LIN {X 0,Y 156.814,Z 593.588,A -85,B 0,C 180,E1 -25031.921,E2 -25031.921} C_VEL
LIN {X 0,Y 150.311,Z 600.724,A -85,B 0,C 180,E1 -25035.498,E2 -25035.498} C_VEL
LIN {X 0,Y 145.203,Z 605.623,A -85,B 0,C 180,E1 -25038.8,E2 -25038.8} C_VEL
LIN {X 0,Y 138.955,Z 610.891,A -85,B 0,C 180,E1 -25043.868,E2 -25043.868} C_VEL
LIN {X 0,Y 135.035,Z 613.658,A -85,B 0,C 180,E1 -25047.932,E2 -25047.932} C_VEL
LIN {X 0,Y 131.858,Z 615.519,A -85,B 0,C 180,E1 -25052.209,E2 -25052.209} C_VEL
LIN {X 0,Y 129.32,Z 616.538,A -85,B 0,C 180,E1 -25056.713,E2 -25056.713} C_VEL
LIN {X 0,Y 127.481,Z 616.693,A -85,B 0,C 180,E1 -25061.42,E2 -25061.42} C_VEL
LIN {X 0,Y 126.047,Z 615.481,A -85,B 0,C 180,E1 -25067.999,E2 -25067.999} C_VEL
LIN {X 0,Y 125.854,Z 612.811,A -85,B 0,C 180,E1 -25074.097,E2 -25074.097} C_VEL
LIN {X 0,Y 126.43,Z 610.019,A -85,B 0,C 180,E1 -25078.395,E2 -25078.395} C_VEL
LIN {X 0,Y 127.613,Z 605.119,A -85,B 0,C 180,E1 -25083.855,E2 -25083.855} C_VEL
LIN {X 0,Y 129.275,Z 599.296,A -85,B 0,C 180,E1 -25088.733,E2 -25088.733} C_VEL
LIN {X 0,Y 131.792,Z 591.532,A -85,B 0,C 180,E1 -25093.717,E2 -25093.717} C_VEL
LIN {X 0,Y 134.655,Z 582.904,A -85,B 0,C 180,E1 -25097.946,E2 -25097.946} C_VEL
LIN {X 0,Y 137.776,Z 573.446,A -85,B 0,C 180,E1 -25101.563,E2 -25101.563} C_VEL
LIN {X 0,Y 140.914,Z 563.091,A -85,B 0,C 180,E1 -25104.647,E2 -25104.647} C_VEL
LIN {X 0,Y 143.932,Z 551.949,A -85,B 0,C 180,E1 -25107.198,E2 -25107.198} C_VEL
LIN {X 0,Y 146.787,Z 539.398,A -85,B 0,C 180,E1 -25109.38,E2 -25109.38} C_VEL
LIN {X 0,Y 149.013,Z 526.448,A -85,B 0,C 180,E1 -25111.001,E2 -25111.001} C_VEL
LIN {X 0,Y 150.791,Z 512.614,A -85,B 0,C 180,E1 -25112.147,E2 -25112.147} C_VEL
LIN {X 0,Y 154.321,Z 464.5,A -85,B 0,C 180,E1 -25114.472,E2 -25114.472} C_VEL
LIN {X 0,Y 151.514,Z 456.717,A -85,B 0,C 180,E1 -25115.652,E2 -25115.652} C_VEL
LIN {X 0,Y 145.99,Z 443.962,A -85,B 0,C 180,E1 -25117.978,E2 -25117.978} C_VEL
LIN {X 0,Y 136.343,Z 427.063,A -85,B 0,C 180,E1 -25122.154,E2 -25122.154} C_VEL
LIN {X 0,Y 133.91,Z 423.355,A -85,B 0,C 180,E1 -25123.296,E2 -25123.296} C_VEL
LIN {X 0,Y 131.689,Z 419.888,A -85,B 0,C 180,E1 -25124.377,E2 -25124.377} C_VEL
LIN {X 0,Y 129.747,Z 417.326,A -85,B 0,C 180,E1 -25125.327,E2 -25125.327} C_VEL
LIN {X 0,Y 129.207,Z 415.394,A -85,B 0,C 180,E1 -25125.777,E2 -25125.777} C_VEL
LIN {X 0,Y 129.159,Z 415.379,A -85,B 0,C 180,E1 -25129.051,E2 -25129.051} C_VEL
LIN {X 0,Y 129.107,Z 415.403,A -85,B 0,C 180,E1 -25132.394,E2 -25132.394} C_VEL
LIN {X 0,Y 129.12,Z 415.555,A -85,B 0,C 180,E1 -25138.437,E2 -25138.437} C_VEL
LIN {X 0,Y 141.163,Z 449.103,A -85,B 0,C 180,E1 -25142.935,E2 -25142.935} C_VEL
LIN {X 0,Y 142.539,Z 453.928,A -85,B 0,C 180,E1 -25143.477,E2 -25143.477} C_VEL
LIN {X 0,Y 138.064,Z 512.835,A -85,B 0,C 180,E1 -25147.853,E2 -25147.853} C_VEL
LIN {X 0,Y 136.81,Z 526.19,A -85,B 0,C 180,E1 -25149.363,E2 -25149.363} C_VEL
LIN {X 0,Y 135.038,Z 539.905,A -85,B 0,C 180,E1 -25151.57,E2 -25151.57} C_VEL
LIN {X 0,Y 133.267,Z 551.828,A -85,B 0,C 180,E1 -25154.123,E2 -25154.123} C_VEL
LIN {X 0,Y 131.313,Z 563.456,A -85,B 0,C 180,E1 -25157.328,E2 -25157.328} C_VEL
LIN {X 0,Y 129.648,Z 573.756,A -85,B 0,C 180,E1 -25160.937,E2 -25160.937} C_VEL
LIN {X 0,Y 128.192,Z 583.694,A -85,B 0,C 180,E1 -25165.314,E2 -25165.314} C_VEL
LIN {X 0,Y 127.16,Z 592.452,A -85,B 0,C 180,E1 -25170.17,E2 -25170.17} C_VEL
LIN {X 0,Y 126.587,Z 598.713,A -85,B 0,C 180,E1 -25174.515,E2 -25174.515} C_VEL
LIN {X 0,Y 126.242,Z 603.697,A -85,B 0,C 180,E1 -25178.785,E2 -25178.785} C_VEL
LIN {X 0,Y 126.536,Z 608.396,A -85,B 0,C 180,E1 -25183.876,E2 -25183.876} C_VEL
LIN {X 0,Y 127.673,Z 611.966,A -85,B 0,C 180,E1 -25188.891,E2 -25188.891} C_VEL
LIN {X 0,Y 129.652,Z 614.508,A -85,B 0,C 180,E1 -25193.776,E2 -25193.776} C_VEL
LIN {X 0,Y 133.699,Z 616.42,A -85,B 0,C 180,E1 -25200,E2 -25200} C_VEL
LIN {X 0,Y 136.366,Z 616.802,A -85,B 0,C 180,E1 -25202.954,E2 -25202.954} C_VEL
LIN {X 0,Y 141.861,Z 616.494,A -85,B 0,C 180,E1 -25207.798,E2 -25207.798} C_VEL
LIN {X 0,Y 146.515,Z 615.477,A -85,B 0,C 180,E1 -25211.062,E2 -25211.062} C_VEL
LIN {X 0,Y 152.429,Z 613.559,A -85,B 0,C 180,E1 -25214.495,E2 -25214.495} C_VEL
LIN {X 0,Y 159.649,Z 610.415,A -85,B 0,C 180,E1 -25217.948,E2 -25217.948} C_VEL
LIN {X 0,Y 167.163,Z 606.309,A -85,B 0,C 180,E1 -25220.938,E2 -25220.938} C_VEL
LIN {X 0,Y 175.327,Z 600.967,A -85,B 0,C 180,E1 -25223.631,E2 -25223.631} C_VEL
LIN {X 0,Y 183.895,Z 594.271,A -85,B 0,C 180,E1 -25226.072,E2 -25226.072} C_VEL
LIN {X 0,Y 191.851,Z 586.996,A -85,B 0,C 180,E1 -25228.006,E2 -25228.006} C_VEL
LIN {X 0,Y 200.929,Z 577.067,A -85,B 0,C 180,E1 -25229.954,E2 -25229.954} C_VEL
LIN {X 0,Y 208.869,Z 566.785,A -85,B 0,C 180,E1 -25231.436,E2 -25231.436} C_VEL
LIN {X 0,Y 215.861,Z 555.807,A -85,B 0,C 180,E1 -25232.604,E2 -25232.604} C_VEL
LIN {X 0,Y 222.008,Z 544.013,A -85,B 0,C 180,E1 -25233.573,E2 -25233.573} C_VEL
LIN {X 0,Y 222.564,Z 542.783,A -85,B 0,C 180,E1 -25233.661,E2 -25233.661} C_VEL
LIN {X 0,Y 222.26,Z 543.527,A -85,B 0,C 180,E1 -25234.024,E2 -25234.024} C_VEL
LIN {X 0,Y 216.111,Z 555.561,A -85,B 0,C 180,E1 -25234.806,E2 -25234.806} C_VEL
LIN {X 0,Y 209.059,Z 566.785,A -85,B 0,C 180,E1 -25235.81,E2 -25235.81} C_VEL
LIN {X 0,Y 202.204,Z 576.047,A -85,B 0,C 180,E1 -25236.931,E2 -25236.931} C_VEL
LIN {X 0,Y 193.406,Z 586.164,A -85,B 0,C 180,E1 -25238.628,E2 -25238.628} C_VEL
LIN {X 0,Y 184.852,Z 594.451,A -85,B 0,C 180,E1 -25240.506,E2 -25240.506} C_VEL
LIN {X 0,Y 176.702,Z 601.316,A -85,B 0,C 180,E1 -25242.63,E2 -25242.63} C_VEL
LIN {X 0,Y 168.919,Z 606.927,A -85,B 0,C 180,E1 -25244.989,E2 -25244.989} C_VEL
LIN {X 0,Y 161.618,Z 611.497,A -85,B 0,C 180,E1 -25247.627,E2 -25247.627} C_VEL
LIN {X 0,Y 154.838,Z 615.091,A -85,B 0,C 180,E1 -25250.551,E2 -25250.551} C_VEL
LIN {X 0,Y 150.47,Z 617.021,A -85,B 0,C 180,E1 -25252.618,E2 -25252.618} C_VEL
LIN {X 0,Y 147.428,Z 618.263,A -85,B 0,C 180,E1 -25254.455,E2 -25254.455} C_VEL
LIN {X 0,Y 143.899,Z 619.387,A -85,B 0,C 180,E1 -25256.266,E2 -25256.266} C_VEL
LIN {X 0,Y 136.832,Z 620.603,A -85,B 0,C 180,E1 -25259.067,E2 -25259.067} C_VEL
LIN {X 0,Y 130.119,Z 620.995,A -85,B 0,C 180,E1 -25262.194,E2 -25262.194} C_VEL
LIN {X 0,Y 127.253,Z 620.827,A -85,B 0,C 180,E1 -25264.49,E2 -25264.49} C_VEL
LIN {X 0,Y 123.427,Z 619.799,A -85,B 0,C 180,E1 -25270.028,E2 -25270.028} C_VEL
LIN {X 0,Y 120.931,Z 617.355,A -85,B 0,C 180,E1 -25276.562,E2 -25276.562} C_VEL
LIN {X 0,Y 120.209,Z 614.9,A -85,B 0,C 180,E1 -25281.176,E2 -25281.176} C_VEL
LIN {X 0,Y 119.431,Z 618.676,A -85,B 0,C 180,E1 -25286.631,E2 -25286.631} C_VEL
LIN {X 0,Y 119.476,Z 620.387,A -85,B 0,C 180,E1 -25290.004,E2 -25290.004} C_VEL
LIN {X 0,Y 119.304,Z 621.641,A -85,B 0,C 180,E1 -25293.381,E2 -25293.381} C_VEL
LIN {X 0,Y 119.439,Z 622.507,A -85,B 0,C 180,E1 -25296.763,E2 -25296.763} C_VEL
LIN {X 0,Y 119.838,Z 622.991,A -85,B 0,C 180,E1 -25300.138,E2 -25300.138} C_VEL
LIN {X 0,Y 121.717,Z 622.767,A -85,B 0,C 180,E1 -25306.785,E2 -25306.785} C_VEL
LIN {X 0,Y 125.178,Z 621.049,A -85,B 0,C 180,E1 -25313.146,E2 -25313.146} C_VEL
LIN {X 0,Y 127.591,Z 619.629,A -85,B 0,C 180,E1 -25316.15,E2 -25316.15} C_VEL
LIN {X 0,Y 131.728,Z 616.701,A -85,B 0,C 180,E1 -25320.458,E2 -25320.458} C_VEL
LIN {X 0,Y 137.161,Z 612.307,A -85,B 0,C 180,E1 -25324.933,E2 -25324.933} C_VEL
LIN {X 0,Y 142.046,Z 607.849,A -85,B 0,C 180,E1 -25328.208,E2 -25328.208} C_VEL
LIN {X 0,Y 149.328,Z 600.561,A -85,B 0,C 180,E1 -25332.122,E2 -25332.122} C_VEL
LIN {X 0,Y 153.747,Z 595.518,A -85,B 0,C 180,E1 -25334.199,E2 -25334.199} C_VEL
LIN {X 0,Y 160.891,Z 586.516,A -85,B 0,C 180,E1 -25337.031,E2 -25337.031} C_VEL
LIN {X 0,Y 167.094,Z 577.291,A -85,B 0,C 180,E1 -25339.212,E2 -25339.212} C_VEL
LIN {X 0,Y 172.958,Z 567.158,A -85,B 0,C 180,E1 -25341.003,E2 -25341.003} C_VEL
LIN {X 0,Y 178.353,Z 556.104,A -85,B 0,C 180,E1 -25342.473,E2 -25342.473} C_VEL
LIN {X 0,Y 182.884,Z 544.76,A -85,B 0,C 180,E1 -25343.576,E2 -25343.576} C_VEL
LIN {X 0,Y 187.001,Z 531.214,A -85,B 0,C 180,E1 -25344.489,E2 -25344.489} C_VEL
LIN {X 0,Y 189.733,Z 518.058,A -85,B 0,C 180,E1 -25345.131,E2 -25345.131} C_VEL
LIN {X 0,Y 191.778,Z 501.436,A -85,B 0,C 180,E1 -25345.734,E2 -25345.734} C_VEL
LIN {X 0,Y 189.87,Z 495.263,A -85,B 0,C 180,E1 -25348.362,E2 -25348.362} C_VEL
LIN {X 0,Y 188.453,Z 491.161,A -85,B 0,C 180,E1 -25350.723,E2 -25350.723} C_VEL
LIN {X 0,Y 187.457,Z 488.373,A -85,B 0,C 180,E1 -25352.715,E2 -25352.715} C_VEL
LIN {X 0,Y 186.256,Z 484.816,A -85,B 0,C 180,E1 -25356.257,E2 -25356.257} C_VEL
LIN {X 0,Y 185.612,Z 483.238,A -85,B 0,C 180,E1 -25360.662,E2 -25360.662} C_VEL
LIN {X 0,Y 185.868,Z 483.1,A -85,B 0,C 180,E1 -25363.776,E2 -25363.776} C_VEL
LIN {X 0,Y 186.518,Z 483.864,A -85,B 0,C 180,E1 -25366.553,E2 -25366.553} C_VEL
LIN {X 0,Y 188.505,Z 487.67,A -85,B 0,C 180,E1 -25371.153,E2 -25371.153} C_VEL
LIN {X 0,Y 189.681,Z 490.329,A -85,B 0,C 180,E1 -25373.087,E2 -25373.087} C_VEL
LIN {X 0,Y 191.615,Z 495.259,A -85,B 0,C 180,E1 -25375.793,E2 -25375.793} C_VEL
LIN {X 0,Y 192.192,Z 497.285,A -85,B 0,C 180,E1 -25376.561,E2 -25376.561} C_VEL
LIN {X 0,Y 189.577,Z 517.305,A -85,B 0,C 180,E1 -25377.302,E2 -25377.302} C_VEL
LIN {X 0,Y 186.925,Z 529.37,A -85,B 0,C 180,E1 -25377.949,E2 -25377.949} C_VEL
LIN {X 0,Y 183.131,Z 541.932,A -85,B 0,C 180,E1 -25378.975,E2 -25378.975} C_VEL
LIN {X 0,Y 178.307,Z 553.972,A -85,B 0,C 180,E1 -25380.295,E2 -25380.295} C_VEL
LIN {X 0,Y 172.712,Z 565.3,A -85,B 0,C 180,E1 -25381.994,E2 -25381.994} C_VEL
LIN {X 0,Y 166.225,Z 576.087,A -85,B 0,C 180,E1 -25384.157,E2 -25384.157} C_VEL
LIN {X 0,Y 159.417,Z 585.634,A -85,B 0,C 180,E1 -25386.727,E2 -25386.727} C_VEL
LIN {X 0,Y 153.191,Z 593.177,A -85,B 0,C 180,E1 -25389.463,E2 -25389.463} C_VEL
LIN {X 0,Y 146.117,Z 600.525,A -85,B 0,C 180,E1 -25393.082,E2 -25393.082} C_VEL
LIN {X 0,Y 139.659,Z 606.297,A -85,B 0,C 180,E1 -25397.024,E2 -25397.024} C_VEL
LIN {X 0,Y 133.733,Z 610.924,A -85,B 0,C 180,E1 -25401.585,E2 -25401.585} C_VEL
LIN {X 0,Y 129.384,Z 613.751,A -85,B 0,C 180,E1 -25405.757,E2 -25405.757} C_VEL
LIN {X 0,Y 125.851,Z 615.651,A -85,B 0,C 180,E1 -25410.172,E2 -25410.172} C_VEL
LIN {X 0,Y 122.224,Z 616.902,A -85,B 0,C 180,E1 -25416.382,E2 -25416.382} C_VEL
LIN {X 0,Y 120.535,Z 616.869,A -85,B 0,C 180,E1 -25420.707,E2 -25420.707} C_VEL
LIN {X 0,Y 119.401,Z 616.207,A -85,B 0,C 180,E1 -25425.058,E2 -25425.058} C_VEL
LIN {X 0,Y 118.77,Z 614.548,A -85,B 0,C 180,E1 -25430.287,E2 -25430.287} C_VEL
LIN {X 0,Y 118.922,Z 611.712,A -85,B 0,C 180,E1 -25435.83,E2 -25435.83} C_VEL
LIN {X 0,Y 119.88,Z 607.47,A -85,B 0,C 180,E1 -25441.569,E2 -25441.569} C_VEL
LIN {X 0,Y 121.091,Z 603.118,A -85,B 0,C 180,E1 -25446.025,E2 -25446.025} C_VEL
LIN {X 0,Y 123.43,Z 595.824,A -85,B 0,C 180,E1 -25451.746,E2 -25451.746} C_VEL
LIN {X 0,Y 126.024,Z 588.235,A -85,B 0,C 180,E1 -25456.286,E2 -25456.286} C_VEL
LIN {X 0,Y 129.3,Z 578.829,A -85,B 0,C 180,E1 -25460.611,E2 -25460.611} C_VEL
LIN {X 0,Y 132.902,Z 568.23,A -85,B 0,C 180,E1 -25464.342,E2 -25464.342} C_VEL
LIN {X 0,Y 136.29,Z 556.734,A -85,B 0,C 180,E1 -25467.41,E2 -25467.41} C_VEL
LIN {X 0,Y 139.329,Z 544.864,A -85,B 0,C 180,E1 -25469.816,E2 -25469.816} C_VEL
LIN {X 0,Y 141.868,Z 532.453,A -85,B 0,C 180,E1 -25471.665,E2 -25471.665} C_VEL
LIN {X 0,Y 143.925,Z 519.093,A -85,B 0,C 180,E1 -25473.06,E2 -25473.06} C_VEL
LIN {X 0,Y 145.312,Z 505.915,A -85,B 0,C 180,E1 -25473.904,E2 -25473.904} C_VEL
LIN {X 0,Y 148.25,Z 466.168,A -85,B 0,C 180,E1 -25475.846,E2 -25475.846} C_VEL
LIN {X 0,Y 145.545,Z 458.81,A -85,B 0,C 180,E1 -25477.066,E2 -25477.066} C_VEL
LIN {X 0,Y 140.683,Z 447.539,A -85,B 0,C 180,E1 -25479.23,E2 -25479.23} C_VEL
LIN {X 0,Y 131.73,Z 431.666,A -85,B 0,C 180,E1 -25483.393,E2 -25483.393} C_VEL
LIN {X 0,Y 127.258,Z 424.838,A -85,B 0,C 180,E1 -25485.658,E2 -25485.658} C_VEL
LIN {X 0,Y 125.022,Z 421.328,A -85,B 0,C 180,E1 -25486.882,E2 -25486.882} C_VEL
LIN {X 0,Y 122.82,Z 418.627,A -85,B 0,C 180,E1 -25488.085,E2 -25488.085} C_VEL
LIN {X 0,Y 122.115,Z 416.257,A -85,B 0,C 180,E1 -25488.668,E2 -25488.668} C_VEL
LIN {X 0,Y 121.981,Z 416.289,A -85,B 0,C 180,E1 -25493.78,E2 -25493.78} C_VEL
LIN {X 0,Y 122.048,Z 416.254,A -85,B 0,C 180,E1 -25497.309,E2 -25497.309} C_VEL
LIN {X 0,Y 133.799,Z 449.097,A -85,B 0,C 180,E1 -25502.037,E2 -25502.037} C_VEL
LIN {X 0,Y 135.623,Z 455.022,A -85,B 0,C 180,E1 -25502.769,E2 -25502.769} C_VEL
LIN {X 0,Y 131.049,Z 513.271,A -85,B 0,C 180,E1 -25507.324,E2 -25507.324} C_VEL
LIN {X 0,Y 129.99,Z 524.796,A -85,B 0,C 180,E1 -25508.686,E2 -25508.686} C_VEL
LIN {X 0,Y 128.497,Z 536.585,A -85,B 0,C 180,E1 -25510.57,E2 -25510.57} C_VEL
LIN {X 0,Y 126.561,Z 549.342,A -85,B 0,C 180,E1 -25513.289,E2 -25513.289} C_VEL
LIN {X 0,Y 124.67,Z 560.416,A -85,B 0,C 180,E1 -25516.324,E2 -25516.324} C_VEL
LIN {X 0,Y 122.907,Z 570.872,A -85,B 0,C 180,E1 -25519.962,E2 -25519.962} C_VEL
LIN {X 0,Y 121.489,Z 580.414,A -85,B 0,C 180,E1 -25524.077,E2 -25524.077} C_VEL
LIN {X 0,Y 120.411,Z 588.391,A -85,B 0,C 180,E1 -25528.311,E2 -25528.311} C_VEL
LIN {X 0,Y 119.777,Z 595.461,A -85,B 0,C 180,E1 -25532.951,E2 -25532.951} C_VEL
LIN {X 0,Y 119.289,Z 601.03,A -85,B 0,C 180,E1 -25537.483,E2 -25537.483} C_VEL
LIN {X 0,Y 119.401,Z 606.365,A -85,B 0,C 180,E1 -25542.884,E2 -25542.884} C_VEL
LIN {X 0,Y 120.361,Z 610.464,A -85,B 0,C 180,E1 -25548.207,E2 -25548.207} C_VEL
LIN {X 0,Y 122.226,Z 613.502,A -85,B 0,C 180,E1 -25553.396,E2 -25553.396} C_VEL
LIN {X 0,Y 126.189,Z 616.066,A -85,B 0,C 180,E1 -25560,E2 -25560} C_VEL
LIN {X 0,Y 131.912,Z 617.082,A -85,B 0,C 180,E1 -25566.117,E2 -25566.117} C_VEL
LIN {X 0,Y 139.126,Z 616.472,A -85,B 0,C 180,E1 -25571.657,E2 -25571.657} C_VEL
LIN {X 0,Y 145.979,Z 614.829,A -85,B 0,C 180,E1 -25575.675,E2 -25575.675} C_VEL
LIN {X 0,Y 155.043,Z 611.515,A -85,B 0,C 180,E1 -25579.875,E2 -25579.875} C_VEL
LIN {X 0,Y 162.917,Z 607.693,A -85,B 0,C 180,E1 -25582.845,E2 -25582.845} C_VEL
LIN {X 0,Y 172.28,Z 602.054,A -85,B 0,C 180,E1 -25585.756,E2 -25585.756} C_VEL
LIN {X 0,Y 181.7,Z 595.202,A -85,B 0,C 180,E1 -25588.233,E2 -25588.233} C_VEL
LIN {X 0,Y 189.685,Z 588.324,A -85,B 0,C 180,E1 -25590.012,E2 -25590.012} C_VEL
LIN {X 0,Y 198.209,Z 579.749,A -85,B 0,C 180,E1 -25591.687,E2 -25591.687} C_VEL
LIN {X 0,Y 206.062,Z 570.294,A -85,B 0,C 180,E1 -25593.072,E2 -25593.072} C_VEL
LIN {X 0,Y 208.805,Z 566.622,A -85,B 0,C 180,E1 -25593.5,E2 -25593.5} C_VEL
LIN {X 0,Y 207.576,Z 568.399,A -85,B 0,C 180,E1 -25593.957,E2 -25593.957} C_VEL
LIN {X 0,Y 199.772,Z 578.209,A -85,B 0,C 180,E1 -25595.127,E2 -25595.127} C_VEL
LIN {X 0,Y 190.715,Z 587.823,A -85,B 0,C 180,E1 -25596.731,E2 -25596.731} C_VEL
LIN {X 0,Y 181.924,Z 595.794,A -85,B 0,C 180,E1 -25598.535,E2 -25598.535} C_VEL
LIN {X 0,Y 172.098,Z 603.249,A -85,B 0,C 180,E1 -25600.937,E2 -25600.937} C_VEL
LIN {X 0,Y 162.916,Z 609.165,A -85,B 0,C 180,E1 -25603.647,E2 -25603.647} C_VEL
LIN {X 0,Y 154.129,Z 613.831,A -85,B 0,C 180,E1 -25606.85,E2 -25606.85} C_VEL
LIN {X 0,Y 144.913,Z 617.626,A -85,B 0,C 180,E1 -25610.92,E2 -25610.92} C_VEL
LIN {X 0,Y 137.256,Z 619.942,A -85,B 0,C 180,E1 -25615.725,E2 -25615.725} C_VEL
LIN {X 0,Y 130.568,Z 620.932,A -85,B 0,C 180,E1 -25621.029,E2 -25621.029} C_VEL
LIN {X 0,Y 127.253,Z 620.827,A -85,B 0,C 180,E1 -25624.49,E2 -25624.49} C_VEL
LIN {X 0,Y 124.677,Z 620.452,A -85,B 0,C 180,E1 -25626.9,E2 -25626.9} C_VEL
LIN {X 0,Y 119.438,Z 619.045,A -85,B 0,C 180,E1 -25630.794,E2 -25630.794} C_VEL
LIN {X 0,Y 115.685,Z 617.3,A -85,B 0,C 180,E1 -25634.103,E2 -25634.103} C_VEL
LIN {X 0,Y 113.936,Z 615.773,A -85,B 0,C 180,E1 -25636.82,E2 -25636.82} C_VEL
LIN {X 0,Y 113.674,Z 615.204,A -85,B 0,C 180,E1 -25637.77,E2 -25637.77} C_VEL
LIN {X 0,Y 113.289,Z 613.934,A -85,B 0,C 180,E1 -25640.407,E2 -25640.407} C_VEL
LIN {X 0,Y 112.375,Z 618.036,A -85,B 0,C 180,E1 -25646.419,E2 -25646.419} C_VEL
LIN {X 0,Y 112.409,Z 619.874,A -85,B 0,C 180,E1 -25650.005,E2 -25650.005} C_VEL
LIN {X 0,Y 112.235,Z 621.206,A -85,B 0,C 180,E1 -25653.595,E2 -25653.595} C_VEL
LIN {X 0,Y 112.401,Z 622.138,A -85,B 0,C 180,E1 -25657.188,E2 -25657.188} C_VEL
LIN {X 0,Y 113.665,Z 622.864,A -85,B 0,C 180,E1 -25664.324,E2 -25664.324} C_VEL
LIN {X 0,Y 114.915,Z 622.665,A -85,B 0,C 180,E1 -25667.81,E2 -25667.81} C_VEL
LIN {X 0,Y 118.668,Z 621.097,A -85,B 0,C 180,E1 -25674.497,E2 -25674.497} C_VEL
LIN {X 0,Y 124.107,Z 618.021,A -85,B 0,C 180,E1 -25680.645,E2 -25680.645} C_VEL
LIN {X 0,Y 129.717,Z 614.113,A -85,B 0,C 180,E1 -25685.424,E2 -25685.424} C_VEL
LIN {X 0,Y 136.57,Z 608.514,A -85,B 0,C 180,E1 -25690.04,E2 -25690.04} C_VEL
LIN {X 0,Y 144.192,Z 601.473,A -85,B 0,C 180,E1 -25693.996,E2 -25693.996} C_VEL
LIN {X 0,Y 148.797,Z 596.599,A -85,B 0,C 180,E1 -25696.083,E2 -25696.083} C_VEL
LIN {X 0,Y 156.205,Z 587.88,A -85,B 0,C 180,E1 -25698.909,E2 -25698.909} C_VEL
LIN {X 0,Y 163.305,Z 578.125,A -85,B 0,C 180,E1 -25701.268,E2 -25701.268} C_VEL
LIN {X 0,Y 169.37,Z 568.276,A -85,B 0,C 180,E1 -25703.018,E2 -25703.018} C_VEL
LIN {X 0,Y 174.94,Z 557.509,A -85,B 0,C 180,E1 -25704.446,E2 -25704.446} C_VEL
LIN {X 0,Y 179.778,Z 546.063,A -85,B 0,C 180,E1 -25705.564,E2 -25705.564} C_VEL
LIN {X 0,Y 183.761,Z 534.161,A -85,B 0,C 180,E1 -25706.374,E2 -25706.374} C_VEL
LIN {X 0,Y 186.872,Z 520.734,A -85,B 0,C 180,E1 -25707.062,E2 -25707.062} C_VEL
LIN {X 0,Y 189.048,Z 505.129,A -85,B 0,C 180,E1 -25707.637,E2 -25707.637} C_VEL
LIN {X 0,Y 187.559,Z 499.736,A -85,B 0,C 180,E1 -25710.198,E2 -25710.198} C_VEL
LIN {X 0,Y 186.194,Z 495.329,A -85,B 0,C 180,E1 -25713.067,E2 -25713.067} C_VEL
LIN {X 0,Y 185.049,Z 491.682,A -85,B 0,C 180,E1 -25716.719,E2 -25716.719} C_VEL
LIN {X 0,Y 184.548,Z 490.183,A -85,B 0,C 180,E1 -25721.096,E2 -25721.096} C_VEL
LIN {X 0,Y 185.099,Z 490.392,A -85,B 0,C 180,E1 -25725.25,E2 -25725.25} C_VEL
LIN {X 0,Y 185.432,Z 491.122,A -85,B 0,C 180,E1 -25726.577,E2 -25726.577} C_VEL
LIN {X 0,Y 187.107,Z 494.503,A -85,B 0,C 180,E1 -25730.681,E2 -25730.681} C_VEL
LIN {X 0,Y 188.086,Z 496.935,A -85,B 0,C 180,E1 -25732.415,E2 -25732.415} C_VEL
LIN {X 0,Y 189.497,Z 500.896,A -85,B 0,C 180,E1 -25734.652,E2 -25734.652} C_VEL
LIN {X 0,Y 186.872,Z 519.267,A -85,B 0,C 180,E1 -25735.336,E2 -25735.336} C_VEL
LIN {X 0,Y 183.834,Z 531.923,A -85,B 0,C 180,E1 -25736.057,E2 -25736.057} C_VEL
LIN {X 0,Y 179.308,Z 545.422,A -85,B 0,C 180,E1 -25737.183,E2 -25737.183} C_VEL
LIN {X 0,Y 174.902,Z 555.644,A -85,B 0,C 180,E1 -25738.339,E2 -25738.339} C_VEL
LIN {X 0,Y 169.114,Z 566.643,A -85,B 0,C 180,E1 -25740,E2 -25740} C_VEL
LIN {X 0,Y 162.632,Z 576.798,A -85,B 0,C 180,E1 -25742.028,E2 -25742.028} C_VEL
LIN {X 0,Y 155.961,Z 585.675,A -85,B 0,C 180,E1 -25744.396,E2 -25744.396} C_VEL
LIN {X 0,Y 148.815,Z 593.861,A -85,B 0,C 180,E1 -25747.339,E2 -25747.339} C_VEL
LIN {X 0,Y 141.308,Z 601.174,A -85,B 0,C 180,E1 -25750.985,E2 -25750.985} C_VEL
LIN {X 0,Y 134.158,Z 607.117,A -85,B 0,C 180,E1 -25755.185,E2 -25755.185} C_VEL
LIN {X 0,Y 127.36,Z 611.835,A -85,B 0,C 180,E1 -25760.256,E2 -25760.256} C_VEL
LIN {X 0,Y 123.229,Z 614.255,A -85,B 0,C 180,E1 -25764.135,E2 -25764.135} C_VEL
LIN {X 0,Y 119.737,Z 615.911,A -85,B 0,C 180,E1 -25768.297,E2 -25768.297} C_VEL
LIN {X 0,Y 116.806,Z 616.902,A -85,B 0,C 180,E1 -25772.787,E2 -25772.787} C_VEL
LIN {X 0,Y 114.348,Z 617.17,A -85,B 0,C 180,E1 -25777.924,E2 -25777.924} C_VEL
LIN {X 0,Y 112.61,Z 616.54,A -85,B 0,C 180,E1 -25783.355,E2 -25783.355} C_VEL
LIN {X 0,Y 111.742,Z 614.932,A -85,B 0,C 180,E1 -25789.003,E2 -25789.003} C_VEL
LIN {X 0,Y 111.79,Z 611.797,A -85,B 0,C 180,E1 -25795.536,E2 -25795.536} C_VEL
LIN {X 0,Y 112.607,Z 608.118,A -85,B 0,C 180,E1 -25800.9,E2 -25800.9} C_VEL
LIN {X 0,Y 113.885,Z 603.593,A -85,B 0,C 180,E1 -25805.918,E2 -25805.918} C_VEL
LIN {X 0,Y 116.012,Z 597.087,A -85,B 0,C 180,E1 -25811.451,E2 -25811.451} C_VEL
LIN {X 0,Y 118.578,Z 589.748,A -85,B 0,C 180,E1 -25816.282,E2 -25816.282} C_VEL
LIN {X 0,Y 121.986,Z 580.579,A -85,B 0,C 180,E1 -25820.917,E2 -25820.917} C_VEL
LIN {X 0,Y 125.63,Z 570.27,A -85,B 0,C 180,E1 -25824.879,E2 -25824.879} C_VEL
LIN {X 0,Y 129.046,Z 559.565,A -85,B 0,C 180,E1 -25828.045,E2 -25828.045} C_VEL
LIN {X 0,Y 132.368,Z 547.661,A -85,B 0,C 180,E1 -25830.686,E2 -25830.686} C_VEL
LIN {X 0,Y 135.172,Z 535.332,A -85,B 0,C 180,E1 -25832.727,E2 -25832.727} C_VEL
LIN {X 0,Y 137.333,Z 522.414,A -85,B 0,C 180,E1 -25834.261,E2 -25834.261} C_VEL
LIN {X 0,Y 139.055,Z 508.742,A -85,B 0,C 180,E1 -25835.252,E2 -25835.252} C_VEL
LIN {X 0,Y 142.192,Z 467.652,A -85,B 0,C 180,E1 -25837.351,E2 -25837.351} C_VEL
LIN {X 0,Y 136.265,Z 452.807,A -85,B 0,C 180,E1 -25840.18,E2 -25840.18} C_VEL
LIN {X 0,Y 127.191,Z 436.246,A -85,B 0,C 180,E1 -25844.689,E2 -25844.689} C_VEL
LIN {X 0,Y 122.499,Z 429.181,A -85,B 0,C 180,E1 -25847.233,E2 -25847.233} C_VEL
LIN {X 0,Y 120.267,Z 425.807,A -85,B 0,C 180,E1 -25848.554,E2 -25848.554} C_VEL
LIN {X 0,Y 118.179,Z 422.54,A -85,B 0,C 180,E1 -25849.847,E2 -25849.847} C_VEL
LIN {X 0,Y 115.668,Z 419.453,A -85,B 0,C 180,E1 -25851.416,E2 -25851.416} C_VEL
LIN {X 0,Y 114.98,Z 417.16,A -85,B 0,C 180,E1 -25852.128,E2 -25852.128} C_VEL
LIN {X 0,Y 114.958,Z 417.153,A -85,B 0,C 180,E1 -25856.183,E2 -25856.183} C_VEL
LIN {X 0,Y 125.47,Z 446.337,A -85,B 0,C 180,E1 -25860.71,E2 -25860.71} C_VEL
LIN {X 0,Y 128.567,Z 455.548,A -85,B 0,C 180,E1 -25861.947,E2 -25861.947} C_VEL
LIN {X 0,Y 125.852,Z 491.643,A -85,B 0,C 180,E1 -25864.895,E2 -25864.895} C_VEL
LIN {X 0,Y 123.809,Z 516.474,A -85,B 0,C 180,E1 -25867.12,E2 -25867.12} C_VEL
LIN {X 0,Y 122.263,Z 530.311,A -85,B 0,C 180,E1 -25869.056,E2 -25869.056} C_VEL
LIN {X 0,Y 120.539,Z 542.255,A -85,B 0,C 180,E1 -25871.35,E2 -25871.35} C_VEL
LIN {X 0,Y 118.473,Z 555.108,A -85,B 0,C 180,E1 -25874.613,E2 -25874.613} C_VEL
LIN {X 0,Y 116.499,Z 566.628,A -85,B 0,C 180,E1 -25878.425,E2 -25878.425} C_VEL
LIN {X 0,Y 114.733,Z 577.63,A -85,B 0,C 180,E1 -25883.09,E2 -25883.09} C_VEL
LIN {X 0,Y 113.64,Z 585.464,A -85,B 0,C 180,E1 -25887.238,E2 -25887.238} C_VEL
LIN {X 0,Y 112.894,Z 593.228,A -85,B 0,C 180,E1 -25892.279,E2 -25892.279} C_VEL
LIN {X 0,Y 112.333,Z 599.094,A -85,B 0,C 180,E1 -25896.981,E2 -25896.981} C_VEL
LIN {X 0,Y 112.315,Z 603.999,A -85,B 0,C 180,E1 -25901.767,E2 -25901.767} C_VEL
LIN {X 0,Y 113.102,Z 608.652,A -85,B 0,C 180,E1 -25907.438,E2 -25907.438} C_VEL
LIN {X 0,Y 114.832,Z 612.219,A -85,B 0,C 180,E1 -25912.969,E2 -25912.969} C_VEL
LIN {X 0,Y 118.699,Z 615.421,A -85,B 0,C 180,E1 -25920,E2 -25920} C_VEL
LIN {X 0,Y 124.437,Z 617.107,A -85,B 0,C 180,E1 -25926.486,E2 -25926.486} C_VEL
LIN {X 0,Y 131.779,Z 617.176,A -85,B 0,C 180,E1 -25932.317,E2 -25932.317} C_VEL
LIN {X 0,Y 140.541,Z 615.717,A -85,B 0,C 180,E1 -25937.46,E2 -25937.46} C_VEL
LIN {X 0,Y 145.443,Z 614.346,A -85,B 0,C 180,E1 -25939.77,E2 -25939.77} C_VEL
LIN {X 0,Y 152.14,Z 611.967,A -85,B 0,C 180,E1 -25942.509,E2 -25942.509} C_VEL
LIN {X 0,Y 161.734,Z 607.58,A -85,B 0,C 180,E1 -25945.756,E2 -25945.756} C_VEL
LIN {X 0,Y 170.707,Z 602.438,A -85,B 0,C 180,E1 -25948.259,E2 -25948.259} C_VEL
LIN {X 0,Y 180.059,Z 596.006,A -85,B 0,C 180,E1 -25950.491,E2 -25950.491} C_VEL
LIN {X 0,Y 188.273,Z 589.323,A -85,B 0,C 180,E1 -25952.137,E2 -25952.137} C_VEL
LIN {X 0,Y 193.275,Z 584.705,A -85,B 0,C 180,E1 -25953.055,E2 -25953.055} C_VEL
LIN {X 0,Y 194.444,Z 583.613,A -85,B 0,C 180,E1 -25953.772,E2 -25953.772} C_VEL
LIN {X 0,Y 185.208,Z 592.239,A -85,B 0,C 180,E1 -25955.334,E2 -25955.334} C_VEL
LIN {X 0,Y 174.795,Z 600.35,A -85,B 0,C 180,E1 -25957.436,E2 -25957.436} C_VEL
LIN {X 0,Y 164.833,Z 606.873,A -85,B 0,C 180,E1 -25959.879,E2 -25959.879} C_VEL
LIN {X 0,Y 154.096,Z 612.544,A -85,B 0,C 180,E1 -25963.142,E2 -25963.142} C_VEL
LIN {X 0,Y 144.246,Z 616.634,A -85,B 0,C 180,E1 -25966.996,E2 -25966.996} C_VEL
LIN {X 0,Y 139.495,Z 618.157,A -85,B 0,C 180,E1 -25969.089,E2 -25969.089} C_VEL
LIN {X 0,Y 131.447,Z 620.08,A -85,B 0,C 180,E1 -25973.981,E2 -25973.981} C_VEL
LIN {X 0,Y 124.397,Z 620.679,A -85,B 0,C 180,E1 -25979.443,E2 -25979.443} C_VEL
LIN {X 0,Y 118.84,Z 619.95,A -85,B 0,C 180,E1 -25985.551,E2 -25985.551} C_VEL
LIN {X 0,Y 115.222,Z 617.882,A -85,B 0,C 180,E1 -25992.248,E2 -25992.248} C_VEL
LIN {X 0,Y 113.674,Z 615.204,A -85,B 0,C 180,E1 -25997.77,E2 -25997.77} C_VEL
LIN {X 0,Y 113.024,Z 614.761,A -85,B 0,C 180,E1 -25999.677,E2 -25999.677} C_VEL
LIN {X 0,Y 111.261,Z 615.601,A -85,B 0,C 180,E1 -26002.519,E2 -26002.519} C_VEL
LIN {X 0,Y 106.376,Z 619.062,A -85,B 0,C 180,E1 -26009.292,E2 -26009.292} C_VEL
LIN {X 0,Y 105.244,Z 620.261,A -85,B 0,C 180,E1 -26012.457,E2 -26012.457} C_VEL
LIN {X 0,Y 105.162,Z 620.631,A -85,B 0,C 180,E1 -26013.535,E2 -26013.535} C_VEL
LIN {X 0,Y 105.343,Z 621.757,A -85,B 0,C 180,E1 -26017.673,E2 -26017.673} C_VEL
LIN {X 0,Y 106.792,Z 622.624,A -85,B 0,C 180,E1 -26025.267,E2 -26025.267} C_VEL
LIN {X 0,Y 109.913,Z 622.026,A -85,B 0,C 180,E1 -26032.565,E2 -26032.565} C_VEL
LIN {X 0,Y 114.985,Z 619.883,A -85,B 0,C 180,E1 -26039.278,E2 -26039.278} C_VEL
LIN {X 0,Y 121.453,Z 616.209,A -85,B 0,C 180,E1 -26045.361,E2 -26045.361} C_VEL
LIN {X 0,Y 127.111,Z 612.324,A -85,B 0,C 180,E1 -26049.487,E2 -26049.487} C_VEL
LIN {X 0,Y 133.459,Z 607.38,A -85,B 0,C 180,E1 -26053.208,E2 -26053.208} C_VEL
LIN {X 0,Y 140.344,Z 601.275,A -85,B 0,C 180,E1 -26056.567,E2 -26056.567} C_VEL
LIN {X 0,Y 147.846,Z 593.746,A -85,B 0,C 180,E1 -26059.52,E2 -26059.52} C_VEL
LIN {X 0,Y 155.661,Z 584.432,A -85,B 0,C 180,E1 -26062.201,E2 -26062.201} C_VEL
LIN {X 0,Y 163.176,Z 573.881,A -85,B 0,C 180,E1 -26064.39,E2 -26064.39} C_VEL
LIN {X 0,Y 169.574,Z 563.073,A -85,B 0,C 180,E1 -26065.991,E2 -26065.991} C_VEL
LIN {X 0,Y 175.399,Z 551.068,A -85,B 0,C 180,E1 -26067.297,E2 -26067.297} C_VEL
LIN {X 0,Y 180.033,Z 539.094,A -85,B 0,C 180,E1 -26068.203,E2 -26068.203} C_VEL
LIN {X 0,Y 183.863,Z 525.354,A -85,B 0,C 180,E1 -26068.963,E2 -26068.963} C_VEL
LIN {X 0,Y 186.257,Z 512.053,A -85,B 0,C 180,E1 -26069.487,E2 -26069.487} C_VEL
LIN {X 0,Y 186.638,Z 508.854,A -85,B 0,C 180,E1 -26069.621,E2 -26069.621} C_VEL
LIN {X 0,Y 185.352,Z 504.107,A -85,B 0,C 180,E1 -26072.24,E2 -26072.24} C_VEL
LIN {X 0,Y 184.573,Z 501.195,A -85,B 0,C 180,E1 -26074.448,E2 -26074.448} C_VEL
LIN {X 0,Y 183.884,Z 498.546,A -85,B 0,C 180,E1 -26077.186,E2 -26077.186} C_VEL
LIN {X 0,Y 183.495,Z 497.242,A -85,B 0,C 180,E1 -26080.984,E2 -26080.984} C_VEL
LIN {X 0,Y 183.883,Z 497.265,A -85,B 0,C 180,E1 -26084.482,E2 -26084.482} C_VEL
LIN {X 0,Y 184.2,Z 497.897,A -85,B 0,C 180,E1 -26086.041,E2 -26086.041} C_VEL
LIN {X 0,Y 185.752,Z 501.336,A -85,B 0,C 180,E1 -26090.212,E2 -26090.212} C_VEL
LIN {X 0,Y 186.646,Z 503.936,A -85,B 0,C 180,E1 -26091.974,E2 -26091.974} C_VEL
LIN {X 0,Y 187.06,Z 505.104,A -85,B 0,C 180,E1 -26092.694,E2 -26092.694} C_VEL
LIN {X 0,Y 184.655,Z 520.504,A -85,B 0,C 180,E1 -26093.285,E2 -26093.285} C_VEL
LIN {X 0,Y 181.455,Z 532.972,A -85,B 0,C 180,E1 -26093.994,E2 -26093.994} C_VEL
LIN {X 0,Y 176.804,Z 546.153,A -85,B 0,C 180,E1 -26095.06,E2 -26095.06} C_VEL
LIN {X 0,Y 171.67,Z 557.352,A -85,B 0,C 180,E1 -26096.314,E2 -26096.314} C_VEL
LIN {X 0,Y 165.096,Z 568.992,A -85,B 0,C 180,E1 -26098.099,E2 -26098.099} C_VEL
LIN {X 0,Y 158.694,Z 578.4,A -85,B 0,C 180,E1 -26100,E2 -26100} C_VEL
LIN {X 0,Y 152.411,Z 586.271,A -85,B 0,C 180,E1 -26102.088,E2 -26102.088} C_VEL
LIN {X 0,Y 145.369,Z 593.918,A -85,B 0,C 180,E1 -26104.801,E2 -26104.801} C_VEL
LIN {X 0,Y 138.684,Z 600.163,A -85,B 0,C 180,E1 -26107.766,E2 -26107.766} C_VEL
LIN {X 0,Y 132.458,Z 605.243,A -85,B 0,C 180,E1 -26111.004,E2 -26111.004} C_VEL
LIN {X 0,Y 126.969,Z 609.141,A -85,B 0,C 180,E1 -26114.368,E2 -26114.368} C_VEL
LIN {X 0,Y 121.784,Z 612.342,A -85,B 0,C 180,E1 -26118.195,E2 -26118.195} C_VEL
LIN {X 0,Y 115.533,Z 615.501,A -85,B 0,C 180,E1 -26124.141,E2 -26124.141} C_VEL
LIN {X 0,Y 110.767,Z 617.091,A -85,B 0,C 180,E1 -26130.504,E2 -26130.504} C_VEL
LIN {X 0,Y 107.062,Z 617.276,A -85,B 0,C 180,E1 -26138.019,E2 -26138.019} C_VEL
LIN {X 0,Y 105.58,Z 616.531,A -85,B 0,C 180,E1 -26142.92,E2 -26142.92} C_VEL
LIN {X 0,Y 104.575,Z 614.224,A -85,B 0,C 180,E1 -26150.318,E2 -26150.318} C_VEL
LIN {X 0,Y 104.932,Z 610.455,A -85,B 0,C 180,E1 -26157.595,E2 -26157.595} C_VEL
LIN {X 0,Y 105.766,Z 607.119,A -85,B 0,C 180,E1 -26162.275,E2 -26162.275} C_VEL
LIN {X 0,Y 107.36,Z 601.928,A -85,B 0,C 180,E1 -26167.947,E2 -26167.947} C_VEL
LIN {X 0,Y 109.828,Z 594.981,A -85,B 0,C 180,E1 -26173.715,E2 -26173.715} C_VEL
LIN {X 0,Y 113.154,Z 586.161,A -85,B 0,C 180,E1 -26179.257,E2 -26179.257} C_VEL
LIN {X 0,Y 116.964,Z 576.169,A -85,B 0,C 180,E1 -26183.96,E2 -26183.96} C_VEL
LIN {X 0,Y 120.92,Z 564.987,A -85,B 0,C 180,E1 -26187.914,E2 -26187.914} C_VEL
LIN {X 0,Y 124.224,Z 554.564,A -85,B 0,C 180,E1 -26190.707,E2 -26190.707} C_VEL
LIN {X 0,Y 127.434,Z 542.446,A -85,B 0,C 180,E1 -26193.157,E2 -26193.157} C_VEL
LIN {X 0,Y 130.117,Z 529.787,A -85,B 0,C 180,E1 -26195.031,E2 -26195.031} C_VEL
LIN {X 0,Y 132.078,Z 517.374,A -85,B 0,C 180,E1 -26196.288,E2 -26196.288} C_VEL
LIN {X 0,Y 133.71,Z 500.753,A -85,B 0,C 180,E1 -26197.3,E2 -26197.3} C_VEL
LIN {X 0,Y 136.25,Z 469.303,A -85,B 0,C 180,E1 -26198.925,E2 -26198.925} C_VEL
LIN {X 0,Y 130.83,Z 455.889,A -85,B 0,C 180,E1 -26201.731,E2 -26201.731} C_VEL
LIN {X 0,Y 122.555,Z 440.649,A -85,B 0,C 180,E1 -26206.146,E2 -26206.146} C_VEL
LIN {X 0,Y 116.319,Z 431.034,A -85,B 0,C 180,E1 -26209.897,E2 -26209.897} C_VEL
LIN {X 0,Y 113.505,Z 426.966,A -85,B 0,C 180,E1 -26211.755,E2 -26211.755} C_VEL
LIN {X 0,Y 111.325,Z 423.621,A -85,B 0,C 180,E1 -26213.316,E2 -26213.316} C_VEL
LIN {X 0,Y 108.655,Z 420.398,A -85,B 0,C 180,E1 -26215.278,E2 -26215.278} C_VEL
LIN {X 0,Y 116.521,Z 441.662,A -85,B 0,C 180,E1 -26218.925,E2 -26218.925} C_VEL
LIN {X 0,Y 121.758,Z 457.059,A -85,B 0,C 180,E1 -26221.21,E2 -26221.21} C_VEL
LIN {X 0,Y 117.137,Z 512.701,A -85,B 0,C 180,E1 -26226.096,E2 -26226.096} C_VEL
LIN {X 0,Y 115.884,Z 525.247,A -85,B 0,C 180,E1 -26227.726,E2 -26227.726} C_VEL
LIN {X 0,Y 114.137,Z 537.85,A -85,B 0,C 180,E1 -26230.017,E2 -26230.017} C_VEL
LIN {X 0,Y 112.115,Z 550.442,A -85,B 0,C 180,E1 -26233.098,E2 -26233.098} C_VEL
LIN {X 0,Y 110.161,Z 561.744,A -85,B 0,C 180,E1 -26236.699,E2 -26236.699} C_VEL
LIN {X 0,Y 108.156,Z 573.615,A -85,B 0,C 180,E1 -26241.562,E2 -26241.562} C_VEL
LIN {X 0,Y 106.929,Z 582.266,A -85,B 0,C 180,E1 -26246.035,E2 -26246.035} C_VEL
LIN {X 0,Y 106.036,Z 590.9,A -85,B 0,C 180,E1 -26251.565,E2 -26251.565} C_VEL
LIN {X 0,Y 105.435,Z 596.953,A -85,B 0,C 180,E1 -26256.425,E2 -26256.425} C_VEL
LIN {X 0,Y 105.391,Z 603.127,A -85,B 0,C 180,E1 -26262.537,E2 -26262.537} C_VEL
LIN {X 0,Y 106.313,Z 608.004,A -85,B 0,C 180,E1 -26268.561,E2 -26268.561} C_VEL
LIN {X 0,Y 108.247,Z 611.723,A -85,B 0,C 180,E1 -26274.411,E2 -26274.411} C_VEL
LIN {X 0,Y 112.496,Z 615.255,A -85,B 0,C 180,E1 -26281.839,E2 -26281.839} C_VEL
LIN {X 0,Y 116.953,Z 616.83,A -85,B 0,C 180,E1 -26286.902,E2 -26286.902} C_VEL
LIN {X 0,Y 124.436,Z 617.584,A -85,B 0,C 180,E1 -26293.057,E2 -26293.057} C_VEL
LIN {X 0,Y 133.375,Z 616.827,A -85,B 0,C 180,E1 -26298.431,E2 -26298.431} C_VEL
LIN {X 0,Y 138.364,Z 615.843,A -85,B 0,C 180,E1 -26300.827,E2 -26300.827} C_VEL
LIN {X 0,Y 149.157,Z 612.613,A -85,B 0,C 180,E1 -26305.091,E2 -26305.091} C_VEL
LIN {X 0,Y 157.766,Z 609.068,A -85,B 0,C 180,E1 -26307.797,E2 -26307.797} C_VEL
LIN {X 0,Y 167.286,Z 604.203,A -85,B 0,C 180,E1 -26310.274,E2 -26310.274} C_VEL
LIN {X 0,Y 176.953,Z 598.148,A -85,B 0,C 180,E1 -26312.424,E2 -26312.424} C_VEL
LIN {X 0,Y 181.458,Z 594.911,A -85,B 0,C 180,E1 -26313.298,E2 -26313.298} C_VEL
LIN {X 0,Y 179.793,Z 596.189,A -85,B 0,C 180,E1 -26313.848,E2 -26313.848} C_VEL
LIN {X 0,Y 172.197,Z 601.564,A -85,B 0,C 180,E1 -26315.292,E2 -26315.292} C_VEL
LIN {X 0,Y 163.347,Z 606.913,A -85,B 0,C 180,E1 -26317.26,E2 -26317.26} C_VEL
LIN {X 0,Y 154.849,Z 611.276,A -85,B 0,C 180,E1 -26319.512,E2 -26319.512} C_VEL
LIN {X 0,Y 149.394,Z 613.651,A -85,B 0,C 180,E1 -26321.182,E2 -26321.182} C_VEL
LIN {X 0,Y 139.168,Z 617.264,A -85,B 0,C 180,E1 -26325.014,E2 -26325.014} C_VEL
LIN {X 0,Y 133.526,Z 618.742,A -85,B 0,C 180,E1 -26327.466,E2 -26327.466} C_VEL
LIN {X 0,Y 125.774,Z 620.13,A -85,B 0,C 180,E1 -26332.078,E2 -26332.078} C_VEL
LIN {X 0,Y 118.335,Z 620.37,A -85,B 0,C 180,E1 -26337.694,E2 -26337.694} C_VEL
LIN {X 0,Y 112.431,Z 619.269,A -85,B 0,C 180,E1 -26344.057,E2 -26344.057} C_VEL
LIN {X 0,Y 108.539,Z 616.885,A -85,B 0,C 180,E1 -26351.115,E2 -26351.115} C_VEL
LIN {X 0,Y 106.603,Z 613.082,A -85,B 0,C 180,E1 -26358.598,E2 -26358.598} C_VEL
LIN {X 0,Y 106.504,Z 612.793,A -85,B 0,C 180,E1 -26359.309,E2 -26359.309} C_VEL
LIN {X 0,Y 105.315,Z 617.395,A -85,B 0,C 180,E1 -26366.179,E2 -26366.179} C_VEL
LIN {X 0,Y 105.333,Z 619.301,A -85,B 0,C 180,E1 -26370.005,E2 -26370.005} C_VEL
LIN {X 0,Y 105.162,Z 620.631,A -85,B 0,C 180,E1 -26373.535,E2 -26373.535} C_VEL
LIN {X 0,Y 104.612,Z 621.62,A -85,B 0,C 180,E1 -26376.7,E2 -26376.7} C_VEL
LIN {X 0,Y 102.423,Z 622.466,A -85,B 0,C 180,E1 -26382.037,E2 -26382.037} C_VEL
LIN {X 0,Y 101.107,Z 622.562,A -85,B 0,C 180,E1 -26386.481,E2 -26386.481} C_VEL
LIN {X 0,Y 101.305,Z 622.375,A -85,B 0,C 180,E1 -26389.847,E2 -26389.847} C_VEL
LIN {X 0,Y 101.715,Z 622.271,A -85,B 0,C 180,E1 -26390.941,E2 -26390.941} C_VEL
LIN {X 0,Y 105.894,Z 621.177,A -85,B 0,C 180,E1 -26397.688,E2 -26397.688} C_VEL
LIN {X 0,Y 108.829,Z 620.032,A -85,B 0,C 180,E1 -26401.112,E2 -26401.112} C_VEL
LIN {X 0,Y 115.75,Z 616.521,A -85,B 0,C 180,E1 -26407.39,E2 -26407.39} C_VEL
LIN {X 0,Y 121.725,Z 612.825,A -85,B 0,C 180,E1 -26411.609,E2 -26411.609} C_VEL
LIN {X 0,Y 128.414,Z 608.104,A -85,B 0,C 180,E1 -26415.361,E2 -26415.361} C_VEL
LIN {X 0,Y 136.822,Z 601.136,A -85,B 0,C 180,E1 -26419.263,E2 -26419.263} C_VEL
LIN {X 0,Y 144.736,Z 593.608,A -85,B 0,C 180,E1 -26422.103,E2 -26422.103} C_VEL
LIN {X 0,Y 152.879,Z 584.328,A -85,B 0,C 180,E1 -26424.69,E2 -26424.69} C_VEL
LIN {X 0,Y 160.695,Z 573.854,A -85,B 0,C 180,E1 -26426.77,E2 -26426.77} C_VEL
LIN {X 0,Y 167.286,Z 563.185,A -85,B 0,C 180,E1 -26428.297,E2 -26428.297} C_VEL
LIN {X 0,Y 173.289,Z 551.248,A -85,B 0,C 180,E1 -26429.527,E2 -26429.527} C_VEL
LIN {X 0,Y 177.904,Z 539.734,A -85,B 0,C 180,E1 -26430.359,E2 -26430.359} C_VEL
LIN {X 0,Y 181.724,Z 526.941,A -85,B 0,C 180,E1 -26431.037,E2 -26431.037} C_VEL
LIN {X 0,Y 184.407,Z 512.954,A -85,B 0,C 180,E1 -26431.621,E2 -26431.621} C_VEL
LIN {X 0,Y 183.641,Z 509.416,A -85,B 0,C 180,E1 -26433.83,E2 -26433.83} C_VEL
LIN {X 0,Y 182.778,Z 505.564,A -85,B 0,C 180,E1 -26437.387,E2 -26437.387} C_VEL
LIN {X 0,Y 182.443,Z 504.303,A -85,B 0,C 180,E1 -26440.87,E2 -26440.87} C_VEL
LIN {X 0,Y 182.809,Z 504.279,A -85,B 0,C 180,E1 -26444.389,E2 -26444.389} C_VEL
LIN {X 0,Y 183.045,Z 504.77,A -85,B 0,C 180,E1 -26445.643,E2 -26445.643} C_VEL
LIN {X 0,Y 184.421,Z 508.141,A -85,B 0,C 180,E1 -26449.722,E2 -26449.722} C_VEL
LIN {X 0,Y 184.808,Z 509.599,A -85,B 0,C 180,E1 -26450.698,E2 -26450.698} C_VEL
LIN {X 0,Y 182.225,Z 523.622,A -85,B 0,C 180,E1 -26451.281,E2 -26451.281} C_VEL
LIN {X 0,Y 179.068,Z 534.923,A -85,B 0,C 180,E1 -26451.93,E2 -26451.93} C_VEL
LIN {X 0,Y 174.507,Z 547.149,A -85,B 0,C 180,E1 -26452.897,E2 -26452.897} C_VEL
LIN {X 0,Y 168.928,Z 558.714,A -85,B 0,C 180,E1 -26454.167,E2 -26454.167} C_VEL
LIN {X 0,Y 162.067,Z 570.228,A -85,B 0,C 180,E1 -26455.895,E2 -26455.895} C_VEL
LIN {X 0,Y 154.725,Z 580.26,A -85,B 0,C 180,E1 -26457.931,E2 -26457.931} C_VEL
LIN {X 0,Y 147.597,Z 588.508,A -85,B 0,C 180,E1 -26460.203,E2 -26460.203} C_VEL
LIN {X 0,Y 140.372,Z 595.721,A -85,B 0,C 180,E1 -26462.87,E2 -26462.87} C_VEL
LIN {X 0,Y 132.922,Z 602.081,A -85,B 0,C 180,E1 -26466.07,E2 -26466.07} C_VEL
LIN {X 0,Y 125.994,Z 607.142,A -85,B 0,C 180,E1 -26469.634,E2 -26469.634} C_VEL
LIN {X 0,Y 119.585,Z 611.11,A -85,B 0,C 180,E1 -26473.597,E2 -26473.597} C_VEL
LIN {X 0,Y 111.992,Z 614.941,A -85,B 0,C 180,E1 -26479.714,E2 -26479.714} C_VEL
LIN {X 0,Y 107.818,Z 616.521,A -85,B 0,C 180,E1 -26484.126,E2 -26484.126} C_VEL
LIN {X 0,Y 104.338,Z 617.389,A -85,B 0,C 180,E1 -26488.869,E2 -26488.869} C_VEL
LIN {X 0,Y 101.542,Z 617.625,A -85,B 0,C 180,E1 -26493.836,E2 -26493.836} C_VEL
LIN {X 0,Y 99.307,Z 617.083,A -85,B 0,C 180,E1 -26499.564,E2 -26499.564} C_VEL
LIN {X 0,Y 97.881,Z 615.598,A -85,B 0,C 180,E1 -26505.892,E2 -26505.892} C_VEL
LIN {X 0,Y 97.427,Z 613.053,A -85,B 0,C 180,E1 -26512.514,E2 -26512.514} C_VEL
LIN {X 0,Y 98.169,Z 608.882,A -85,B 0,C 180,E1 -26519.919,E2 -26519.919} C_VEL
LIN {X 0,Y 99.685,Z 603.77,A -85,B 0,C 180,E1 -26526.425,E2 -26526.425} C_VEL
LIN {X 0,Y 102.12,Z 596.952,A -85,B 0,C 180,E1 -26532.939,E2 -26532.939} C_VEL
LIN {X 0,Y 105.03,Z 589.432,A -85,B 0,C 180,E1 -26538.415,E2 -26538.415} C_VEL
LIN {X 0,Y 108.823,Z 580.145,A -85,B 0,C 180,E1 -26543.506,E2 -26543.506} C_VEL
LIN {X 0,Y 112.819,Z 569.848,A -85,B 0,C 180,E1 -26547.777,E2 -26547.777} C_VEL
LIN {X 0,Y 116.72,Z 558.567,A -85,B 0,C 180,E1 -26551.289,E2 -26551.289} C_VEL
LIN {X 0,Y 120.458,Z 545.998,A -85,B 0,C 180,E1 -26554.178,E2 -26554.178} C_VEL
LIN {X 0,Y 123.243,Z 534.405,A -85,B 0,C 180,E1 -26556.134,E2 -26556.134} C_VEL
LIN {X 0,Y 125.715,Z 520.465,A -85,B 0,C 180,E1 -26557.771,E2 -26557.771} C_VEL
LIN {X 0,Y 127.426,Z 506.608,A -85,B 0,C 180,E1 -26558.744,E2 -26558.744} C_VEL
LIN {X 0,Y 130.382,Z 471.197,A -85,B 0,C 180,E1 -26560.639,E2 -26560.639} C_VEL
LIN {X 0,Y 125.807,Z 459.747,A -85,B 0,C 180,E1 -26563.178,E2 -26563.178} C_VEL
LIN {X 0,Y 118.138,Z 445.264,A -85,B 0,C 180,E1 -26567.634,E2 -26567.634} C_VEL
LIN {X 0,Y 112.494,Z 436.371,A -85,B 0,C 180,E1 -26571.274,E2 -26571.274} C_VEL
LIN {X 0,Y 109.421,Z 431.884,A -85,B 0,C 180,E1 -26573.466,E2 -26573.466} C_VEL
LIN {X 0,Y 108.957,Z 431.53,A -85,B 0,C 180,E1 -26573.779,E2 -26573.779} C_VEL
LIN {X 0,Y 107.955,Z 432.216,A -85,B 0,C 180,E1 -26574.297,E2 -26574.297} C_VEL
LIN {X 0,Y 106.31,Z 432.198,A -85,B 0,C 180,E1 -26575.317,E2 -26575.317} C_VEL
LIN {X 0,Y 105.554,Z 431.523,A -85,B 0,C 180,E1 -26575.877,E2 -26575.877} C_VEL
LIN {X 0,Y 114.394,Z 456.787,A -85,B 0,C 180,E1 -26580.138,E2 -26580.138} C_VEL
LIN {X 0,Y 114.864,Z 458.59,A -85,B 0,C 180,E1 -26580.386,E2 -26580.386} C_VEL
LIN {X 0,Y 110.103,Z 513.204,A -85,B 0,C 180,E1 -26585.525,E2 -26585.525} C_VEL
LIN {X 0,Y 108.767,Z 525.789,A -85,B 0,C 180,E1 -26587.29,E2 -26587.29} C_VEL
LIN {X 0,Y 106.892,Z 538.899,A -85,B 0,C 180,E1 -26589.881,E2 -26589.881} C_VEL
LIN {X 0,Y 104.856,Z 551.45,A -85,B 0,C 180,E1 -26593.205,E2 -26593.205} C_VEL
LIN {X 0,Y 102.61,Z 564.094,A -85,B 0,C 180,E1 -26597.662,E2 -26597.662} C_VEL
LIN {X 0,Y 100.867,Z 574.615,A -85,B 0,C 180,E1 -26602.434,E2 -26602.434} C_VEL
LIN {X 0,Y 99.532,Z 584.083,A -85,B 0,C 180,E1 -26607.911,E2 -26607.911} C_VEL
LIN {X 0,Y 98.825,Z 592.022,A -85,B 0,C 180,E1 -26613.61,E2 -26613.61} C_VEL
LIN {X 0,Y 98.373,Z 599.234,A -85,B 0,C 180,E1 -26620.162,E2 -26620.162} C_VEL
LIN {X 0,Y 98.731,Z 604.044,A -85,B 0,C 180,E1 -26625.573,E2 -26625.573} C_VEL
LIN {X 0,Y 100.144,Z 608.683,A -85,B 0,C 180,E1 -26631.931,E2 -26631.931} C_VEL
LIN {X 0,Y 102.679,Z 612.286,A -85,B 0,C 180,E1 -26638.038,E2 -26638.038} C_VEL
LIN {X 0,Y 106.369,Z 614.931,A -85,B 0,C 180,E1 -26643.788,E2 -26643.788} C_VEL
LIN {X 0,Y 113.087,Z 617.172,A -85,B 0,C 180,E1 -26650.745,E2 -26650.745} C_VEL
LIN {X 0,Y 121.499,Z 617.841,A -85,B 0,C 180,E1 -26656.811,E2 -26656.811} C_VEL
LIN {X 0,Y 127.13,Z 617.553,A -85,B 0,C 180,E1 -26659.997,E2 -26659.997} C_VEL
LIN {X 0,Y 136.699,Z 615.995,A -85,B 0,C 180,E1 -26664.286,E2 -26664.286} C_VEL
LIN {X 0,Y 142.322,Z 614.561,A -85,B 0,C 180,E1 -26666.387,E2 -26666.387} C_VEL
LIN {X 0,Y 151.271,Z 611.604,A -85,B 0,C 180,E1 -26669.199,E2 -26669.199} C_VEL
LIN {X 0,Y 160.772,Z 607.543,A -85,B 0,C 180,E1 -26671.639,E2 -26671.639} C_VEL
LIN {X 0,Y 168.292,Z 603.661,A -85,B 0,C 180,E1 -26673.368,E2 -26673.368} C_VEL
LIN {X 0,Y 159.229,Z 608.571,A -85,B 0,C 180,E1 -26675.266,E2 -26675.266} C_VEL
LIN {X 0,Y 150.493,Z 612.476,A -85,B 0,C 180,E1 -26677.455,E2 -26677.455} C_VEL
LIN {X 0,Y 144.864,Z 614.641,A -85,B 0,C 180,E1 -26679.09,E2 -26679.09} C_VEL
LIN {X 0,Y 134.262,Z 617.814,A -85,B 0,C 180,E1 -26682.882,E2 -26682.882} C_VEL
LIN {X 0,Y 127.575,Z 619.173,A -85,B 0,C 180,E1 -26685.738,E2 -26685.738} C_VEL
LIN {X 0,Y 120.254,Z 620.051,A -85,B 0,C 180,E1 -26690,E2 -26690} C_VEL
LIN {X 0,Y 112.401,Z 619.932,A -85,B 0,C 180,E1 -26695.761,E2 -26695.761} C_VEL
LIN {X 0,Y 106.113,Z 618.524,A -85,B 0,C 180,E1 -26702.385,E2 -26702.385} C_VEL
LIN {X 0,Y 101.907,Z 615.77,A -85,B 0,C 180,E1 -26709.835,E2 -26709.835} C_VEL
LIN {X 0,Y 99.747,Z 611.511,A -85,B 0,C 180,E1 -26718.061,E2 -26718.061} C_VEL
LIN {X 0,Y 98.452,Z 615.53,A -85,B 0,C 180,E1 -26723.859,E2 -26723.859} C_VEL
LIN {X 0,Y 98.266,Z 618.698,A -85,B 0,C 180,E1 -26730.005,E2 -26730.005} C_VEL
LIN {X 0,Y 98.089,Z 620.215,A -85,B 0,C 180,E1 -26734.114,E2 -26734.114} C_VEL
LIN {X 0,Y 98.298,Z 621.339,A -85,B 0,C 180,E1 -26738.226,E2 -26738.226} C_VEL
LIN {X 0,Y 98.898,Z 622.062,A -85,B 0,C 180,E1 -26742.315,E2 -26742.315} C_VEL
LIN {X 0,Y 101.41,Z 622.34,A -85,B 0,C 180,E1 -26750.28,E2 -26750.28} C_VEL
LIN {X 0,Y 101.715,Z 622.271,A -85,B 0,C 180,E1 -26750.941,E2 -26750.941} C_VEL
LIN {X 0,Y 102.773,Z 621.948,A -85,B 0,C 180,E1 -26754.196,E2 -26754.196} C_VEL
LIN {X 0,Y 103.588,Z 620.907,A -85,B 0,C 180,E1 -26759.664,E2 -26759.664} C_VEL
LIN {X 0,Y 105.347,Z 619.332,A -85,B 0,C 180,E1 -26764.936,E2 -26764.936} C_VEL
LIN {X 0,Y 107.775,Z 617.999,A -85,B 0,C 180,E1 -26767.734,E2 -26767.734} C_VEL
LIN {X 0,Y 114.323,Z 614.621,A -85,B 0,C 180,E1 -26772.555,E2 -26772.555} C_VEL
LIN {X 0,Y 121.124,Z 610.445,A -85,B 0,C 180,E1 -26776.499,E2 -26776.499} C_VEL
LIN {X 0,Y 128.577,Z 605.16,A -85,B 0,C 180,E1 -26779.934,E2 -26779.934} C_VEL
LIN {X 0,Y 135.049,Z 599.874,A -85,B 0,C 180,E1 -26782.53,E2 -26782.53} C_VEL
LIN {X 0,Y 143.326,Z 592.126,A -85,B 0,C 180,E1 -26785.225,E2 -26785.225} C_VEL
LIN {X 0,Y 151.863,Z 582.62,A -85,B 0,C 180,E1 -26787.633,E2 -26787.633} C_VEL
LIN {X 0,Y 159.227,Z 572.86,A -85,B 0,C 180,E1 -26789.401,E2 -26789.401} C_VEL
LIN {X 0,Y 166.047,Z 561.943,A -85,B 0,C 180,E1 -26790.81,E2 -26790.81} C_VEL
LIN {X 0,Y 172.228,Z 549.799,A -85,B 0,C 180,E1 -26791.943,E2 -26791.943} C_VEL
LIN {X 0,Y 177.219,Z 537.157,A -85,B 0,C 180,E1 -26792.759,E2 -26792.759} C_VEL
LIN {X 0,Y 181.157,Z 523.325,A -85,B 0,C 180,E1 -26793.4,E2 -26793.4} C_VEL
LIN {X 0,Y 182.397,Z 517.272,A -85,B 0,C 180,E1 -26793.645,E2 -26793.645} C_VEL
LIN {X 0,Y 181.872,Z 514.328,A -85,B 0,C 180,E1 -26795.916,E2 -26795.916} C_VEL
LIN {X 0,Y 181.552,Z 512.213,A -85,B 0,C 180,E1 -26798.294,E2 -26798.294} C_VEL
LIN {X 0,Y 181.419,Z 511.149,A -85,B 0,C 180,E1 -26801.946,E2 -26801.946} C_VEL
LIN {X 0,Y 181.849,Z 511.528,A -85,B 0,C 180,E1 -26805.067,E2 -26805.067} C_VEL
LIN {X 0,Y 182.814,Z 514.342,A -85,B 0,C 180,E1 -26808.707,E2 -26808.707} C_VEL
LIN {X 0,Y 179.789,Z 527.798,A -85,B 0,C 180,E1 -26809.251,E2 -26809.251} C_VEL
LIN {X 0,Y 175.641,Z 540.521,A -85,B 0,C 180,E1 -26810.062,E2 -26810.062} C_VEL
LIN {X 0,Y 170.762,Z 551.886,A -85,B 0,C 180,E1 -26811.043,E2 -26811.043} C_VEL
LIN {X 0,Y 164.898,Z 562.734,A -85,B 0,C 180,E1 -26812.285,E2 -26812.285} C_VEL
LIN {X 0,Y 158.16,Z 573.018,A -85,B 0,C 180,E1 -26813.881,E2 -26813.881} C_VEL
LIN {X 0,Y 150.622,Z 582.597,A -85,B 0,C 180,E1 -26815.871,E2 -26815.871} C_VEL
LIN {X 0,Y 142.366,Z 591.356,A -85,B 0,C 180,E1 -26818.385,E2 -26818.385} C_VEL
LIN {X 0,Y 133.588,Z 599.12,A -85,B 0,C 180,E1 -26821.542,E2 -26821.542} C_VEL
LIN {X 0,Y 126.887,Z 604.192,A -85,B 0,C 180,E1 -26824.405,E2 -26824.405} C_VEL
LIN {X 0,Y 117.792,Z 609.995,A -85,B 0,C 180,E1 -26829.132,E2 -26829.132} C_VEL
LIN {X 0,Y 111.82,Z 613.089,A -85,B 0,C 180,E1 -26833.035,E2 -26833.035} C_VEL
LIN {X 0,Y 103.896,Z 616.274,A -85,B 0,C 180,E1 -26839.769,E2 -26839.769} C_VEL
LIN {X 0,Y 99.325,Z 617.488,A -85,B 0,C 180,E1 -26845.122,E2 -26845.122} C_VEL
LIN {X 0,Y 95.592,Z 617.853,A -85,B 0,C 180,E1 -26850.974,E2 -26850.974} C_VEL
LIN {X 0,Y 92.844,Z 617.337,A -85,B 0,C 180,E1 -26857.271,E2 -26857.271} C_VEL
LIN {X 0,Y 90.776,Z 615.383,A -85,B 0,C 180,E1 -26865.822,E2 -26865.822} C_VEL
LIN {X 0,Y 90.417,Z 611.965,A -85,B 0,C 180,E1 -26874.334,E2 -26874.334} C_VEL
LIN {X 0,Y 91.136,Z 608.48,A -85,B 0,C 180,E1 -26880.468,E2 -26880.468} C_VEL
LIN {X 0,Y 92.879,Z 602.937,A -85,B 0,C 180,E1 -26887.763,E2 -26887.763} C_VEL
LIN {X 0,Y 95.172,Z 596.945,A -85,B 0,C 180,E1 -26893.74,E2 -26893.74} C_VEL
LIN {X 0,Y 98.267,Z 589.339,A -85,B 0,C 180,E1 -26899.595,E2 -26899.595} C_VEL
LIN {X 0,Y 102.352,Z 579.778,A -85,B 0,C 180,E1 -26905.071,E2 -26905.071} C_VEL
LIN {X 0,Y 106.68,Z 569.149,A -85,B 0,C 180,E1 -26909.613,E2 -26909.613} C_VEL
LIN {X 0,Y 110.732,Z 557.851,A -85,B 0,C 180,E1 -26913.179,E2 -26913.179} C_VEL
LIN {X 0,Y 114.354,Z 546.178,A -85,B 0,C 180,E1 -26915.925,E2 -26915.925} C_VEL
LIN {X 0,Y 117.289,Z 534.472,A -85,B 0,C 180,E1 -26917.96,E2 -26917.96} C_VEL
LIN {X 0,Y 119.849,Z 520.521,A -85,B 0,C 180,E1 -26919.648,E2 -26919.648} C_VEL
LIN {X 0,Y 121.645,Z 506.676,A -85,B 0,C 180,E1 -26920.632,E2 -26920.632} C_VEL
LIN {X 0,Y 124.561,Z 473.089,A -85,B 0,C 180,E1 -26922.485,E2 -26922.485} C_VEL
LIN {X 0,Y 120.921,Z 463.746,A -85,B 0,C 180,E1 -26924.696,E2 -26924.696} C_VEL
LIN {X 0,Y 113.628,Z 449.575,A -85,B 0,C 180,E1 -26929.313,E2 -26929.313} C_VEL
LIN {X 0,Y 107.756,Z 440.277,A -85,B 0,C 180,E1 -26933.465,E2 -26933.465} C_VEL
LIN {X 0,Y 105.472,Z 443.21,A -85,B 0,C 180,E1 -26934.501,E2 -26934.501} C_VEL
LIN {X 0,Y 104.647,Z 443.747,A -85,B 0,C 180,E1 -26934.957,E2 -26934.957} C_VEL
LIN {X 0,Y 103.043,Z 443.615,A -85,B 0,C 180,E1 -26936.005,E2 -26936.005} C_VEL
LIN {X 0,Y 102.286,Z 442.914,A -85,B 0,C 180,E1 -26936.629,E2 -26936.629} C_VEL
LIN {X 0,Y 107.913,Z 459.373,A -85,B 0,C 180,E1 -26939.455,E2 -26939.455} C_VEL
LIN {X 0,Y 103.142,Z 512.863,A -85,B 0,C 180,E1 -26944.803,E2 -26944.803} C_VEL
LIN {X 0,Y 101.913,Z 524.523,A -85,B 0,C 180,E1 -26946.502,E2 -26946.502} C_VEL
LIN {X 0,Y 99.937,Z 538.07,A -85,B 0,C 180,E1 -26949.259,E2 -26949.259} C_VEL
LIN {X 0,Y 97.917,Z 550.205,A -85,B 0,C 180,E1 -26952.633,E2 -26952.633} C_VEL
LIN {X 0,Y 95.814,Z 562.054,A -85,B 0,C 180,E1 -26956.967,E2 -26956.967} C_VEL
LIN {X 0,Y 93.829,Z 573.711,A -85,B 0,C 180,E1 -26962.512,E2 -26962.512} C_VEL
LIN {X 0,Y 92.58,Z 582.638,A -85,B 0,C 180,E1 -26967.9,E2 -26967.9} C_VEL
LIN {X 0,Y 91.882,Z 590.689,A -85,B 0,C 180,E1 -26973.909,E2 -26973.909} C_VEL
LIN {X 0,Y 91.471,Z 596.97,A -85,B 0,C 180,E1 -26979.772,E2 -26979.772} C_VEL
LIN {X 0,Y 91.936,Z 603.057,A -85,B 0,C 180,E1 -26986.742,E2 -26986.742} C_VEL
LIN {X 0,Y 93.562,Z 607.926,A -85,B 0,C 180,E1 -26993.53,E2 -26993.53} C_VEL
LIN {X 0,Y 96.39,Z 611.704,A -85,B 0,C 180,E1 -27000,E2 -27000} C_VEL
LIN {X 0,Y 102.055,Z 615.357,A -85,B 0,C 180,E1 -27007.916,E2 -27007.916} C_VEL
LIN {X 0,Y 109.783,Z 617.482,A -85,B 0,C 180,E1 -27014.837,E2 -27014.837} C_VEL
LIN {X 0,Y 119.117,Z 618.101,A -85,B 0,C 180,E1 -27020.732,E2 -27020.732} C_VEL
LIN {X 0,Y 124.285,Z 617.862,A -85,B 0,C 180,E1 -27023.318,E2 -27023.318} C_VEL
LIN {X 0,Y 134.695,Z 616.362,A -85,B 0,C 180,E1 -27027.51,E2 -27027.51} C_VEL
LIN {X 0,Y 141.593,Z 614.721,A -85,B 0,C 180,E1 -27029.759,E2 -27029.759} C_VEL
LIN {X 0,Y 151.535,Z 611.536,A -85,B 0,C 180,E1 -27032.46,E2 -27032.46} C_VEL
LIN {X 0,Y 154.347,Z 610.476,A -85,B 0,C 180,E1 -27033.121,E2 -27033.121} C_VEL
LIN {X 0,Y 152.272,Z 611.364,A -85,B 0,C 180,E1 -27033.828,E2 -27033.828} C_VEL
LIN {X 0,Y 140.528,Z 615.504,A -85,B 0,C 180,E1 -27036.859,E2 -27036.859} C_VEL
LIN {X 0,Y 129.558,Z 618.255,A -85,B 0,C 180,E1 -27040.592,E2 -27040.592} C_VEL
LIN {X 0,Y 121.7,Z 619.428,A -85,B 0,C 180,E1 -27043.867,E2 -27043.867} C_VEL
LIN {X 0,Y 114.909,Z 619.895,A -85,B 0,C 180,E1 -27047.725,E2 -27047.725} C_VEL
LIN {X 0,Y 106.617,Z 619.388,A -85,B 0,C 180,E1 -27053.617,E2 -27053.617} C_VEL
LIN {X 0,Y 99.917,Z 617.606,A -85,B 0,C 180,E1 -27060.51,E2 -27060.51} C_VEL
LIN {X 0,Y 95.373,Z 614.579,A -85,B 0,C 180,E1 -27068.386,E2 -27068.386} C_VEL
LIN {X 0,Y 93.022,Z 610.292,A -85,B 0,C 180,E1 -27076.767,E2 -27076.767} C_VEL
LIN {X 0,Y 91.44,Z 614.771,A -85,B 0,C 180,E1 -27083.386,E2 -27083.386} C_VEL
LIN {X 0,Y 91.2,Z 618.095,A -85,B 0,C 180,E1 -27090.006,E2 -27090.006} C_VEL
LIN {X 0,Y 91.029,Z 619.686,A -85,B 0,C 180,E1 -27094.434,E2 -27094.434} C_VEL
LIN {X 0,Y 91.973,Z 621.689,A -85,B 0,C 180,E1 -27103.258,E2 -27103.258} C_VEL
LIN {X 0,Y 94.747,Z 622.175,A -85,B 0,C 180,E1 -27111.776,E2 -27111.776} C_VEL
LIN {X 0,Y 99.657,Z 621.168,A -85,B 0,C 180,E1 -27119.587,E2 -27119.587} C_VEL
LIN {X 0,Y 106.322,Z 618.704,A -85,B 0,C 180,E1 -27126.512,E2 -27126.512} C_VEL
LIN {X 0,Y 107.775,Z 617.999,A -85,B 0,C 180,E1 -27127.734,E2 -27127.734} C_VEL
LIN {X 0,Y 110.419,Z 616.528,A -85,B 0,C 180,E1 -27130.395,E2 -27130.395} C_VEL
LIN {X 0,Y 113.72,Z 613.764,A -85,B 0,C 180,E1 -27134.977,E2 -27134.977} C_VEL
LIN {X 0,Y 117.649,Z 610.515,A -85,B 0,C 180,E1 -27139.168,E2 -27139.168} C_VEL
LIN {X 0,Y 121.11,Z 608.11,A -85,B 0,C 180,E1 -27141.142,E2 -27141.142} C_VEL
LIN {X 0,Y 129.484,Z 602.044,A -85,B 0,C 180,E1 -27144.51,E2 -27144.51} C_VEL
LIN {X 0,Y 138.028,Z 594.845,A -85,B 0,C 180,E1 -27147.161,E2 -27147.161} C_VEL
LIN {X 0,Y 146.756,Z 586.054,A -85,B 0,C 180,E1 -27149.548,E2 -27149.548} C_VEL
LIN {X 0,Y 155.061,Z 576.098,A -85,B 0,C 180,E1 -27151.427,E2 -27151.427} C_VEL
LIN {X 0,Y 162.794,Z 564.856,A -85,B 0,C 180,E1 -27152.93,E2 -27152.93} C_VEL
LIN {X 0,Y 169.104,Z 553.59,A -85,B 0,C 180,E1 -27153.999,E2 -27153.999} C_VEL
LIN {X 0,Y 174.084,Z 542.422,A -85,B 0,C 180,E1 -27154.742,E2 -27154.742} C_VEL
LIN {X 0,Y 178.665,Z 528.818,A -85,B 0,C 180,E1 -27155.401,E2 -27155.401} C_VEL
LIN {X 0,Y 180.414,Z 521.87,A -85,B 0,C 180,E1 -27155.703,E2 -27155.703} C_VEL
LIN {X 0,Y 180.187,Z 519.113,A -85,B 0,C 180,E1 -27158.563,E2 -27158.563} C_VEL
LIN {X 0,Y 180.108,Z 518.148,A -85,B 0,C 180,E1 -27161.81,E2 -27161.81} C_VEL
LIN {X 0,Y 180.45,Z 518.484,A -85,B 0,C 180,E1 -27164.756,E2 -27164.756} C_VEL
LIN {X 0,Y 180.694,Z 520.001,A -85,B 0,C 180,E1 -27166.691,E2 -27166.691} C_VEL
LIN {X 0,Y 177.4,Z 532.319,A -85,B 0,C 180,E1 -27167.22,E2 -27167.22} C_VEL
LIN {X 0,Y 172.363,Z 545.758,A -85,B 0,C 180,E1 -27168.134,E2 -27168.134} C_VEL
LIN {X 0,Y 166.336,Z 557.937,A -85,B 0,C 180,E1 -27169.235,E2 -27169.235} C_VEL
LIN {X 0,Y 159.245,Z 569.302,A -85,B 0,C 180,E1 -27170.714,E2 -27170.714} C_VEL
LIN {X 0,Y 151.764,Z 579.141,A -85,B 0,C 180,E1 -27172.416,E2 -27172.416} C_VEL
LIN {X 0,Y 144.087,Z 587.597,A -85,B 0,C 180,E1 -27174.402,E2 -27174.402} C_VEL
LIN {X 0,Y 135.39,Z 595.65,A -85,B 0,C 180,E1 -27177.025,E2 -27177.025} C_VEL
LIN {X 0,Y 126.513,Z 602.528,A -85,B 0,C 180,E1 -27180.222,E2 -27180.222} C_VEL
LIN {X 0,Y 119.197,Z 607.288,A -85,B 0,C 180,E1 -27183.38,E2 -27183.38} C_VEL
LIN {X 0,Y 111.813,Z 611.327,A -85,B 0,C 180,E1 -27187.222,E2 -27187.222} C_VEL
LIN {X 0,Y 105.131,Z 614.349,A -85,B 0,C 180,E1 -27191.57,E2 -27191.57} C_VEL
LIN {X 0,Y 99.148,Z 616.453,A -85,B 0,C 180,E1 -27196.472,E2 -27196.472} C_VEL
LIN {X 0,Y 92.364,Z 617.908,A -85,B 0,C 180,E1 -27204.052,E2 -27204.052} C_VEL
LIN {X 0,Y 88.883,Z 618.027,A -85,B 0,C 180,E1 -27209.557,E2 -27209.557} C_VEL
LIN {X 0,Y 86.243,Z 617.499,A -85,B 0,C 180,E1 -27215.413,E2 -27215.413} C_VEL
LIN {X 0,Y 84.351,Z 616.21,A -85,B 0,C 180,E1 -27221.802,E2 -27221.802} C_VEL
LIN {X 0,Y 83.315,Z 613.818,A -85,B 0,C 180,E1 -27229.394,E2 -27229.394} C_VEL
LIN {X 0,Y 83.585,Z 610.27,A -85,B 0,C 180,E1 -27237.229,E2 -27237.229} C_VEL
LIN {X 0,Y 85.088,Z 605.01,A -85,B 0,C 180,E1 -27245.601,E2 -27245.601} C_VEL
LIN {X 0,Y 87.316,Z 599.035,A -85,B 0,C 180,E1 -27252.609,E2 -27252.609} C_VEL
LIN {X 0,Y 90.311,Z 592.127,A -85,B 0,C 180,E1 -27258.776,E2 -27258.776} C_VEL
LIN {X 0,Y 94.14,Z 583.454,A -85,B 0,C 180,E1 -27264.64,E2 -27264.64} C_VEL
LIN {X 0,Y 98.397,Z 573.867,A -85,B 0,C 180,E1 -27269.476,E2 -27269.476} C_VEL
LIN {X 0,Y 102.552,Z 563.372,A -85,B 0,C 180,E1 -27273.433,E2 -27273.433} C_VEL
LIN {X 0,Y 106.435,Z 552.459,A -85,B 0,C 180,E1 -27276.498,E2 -27276.498} C_VEL
LIN {X 0,Y 109.928,Z 540.715,A -85,B 0,C 180,E1 -27278.96,E2 -27278.96} C_VEL
LIN {X 0,Y 112.922,Z 527.472,A -85,B 0,C 180,E1 -27280.936,E2 -27280.936} C_VEL
LIN {X 0,Y 115.207,Z 513.568,A -85,B 0,C 180,E1 -27282.278,E2 -27282.278} C_VEL
LIN {X 0,Y 118.939,Z 475.137,A -85,B 0,C 180,E1 -27284.445,E2 -27284.445} C_VEL
LIN {X 0,Y 116.062,Z 467.563,A -85,B 0,C 180,E1 -27286.386,E2 -27286.386} C_VEL
LIN {X 0,Y 109.226,Z 453.959,A -85,B 0,C 180,E1 -27291.083,E2 -27291.083} C_VEL
LIN {X 0,Y 106.805,Z 449.943,A -85,B 0,C 180,E1 -27292.893,E2 -27292.893} C_VEL
LIN {X 0,Y 104.939,Z 450.572,A -85,B 0,C 180,E1 -27293.936,E2 -27293.936} C_VEL
LIN {X 0,Y 102.945,Z 454.182,A -85,B 0,C 180,E1 -27294.745,E2 -27294.745} C_VEL
LIN {X 0,Y 101.326,Z 455.454,A -85,B 0,C 180,E1 -27295.619,E2 -27295.619} C_VEL
LIN {X 0,Y 99.905,Z 455.411,A -85,B 0,C 180,E1 -27296.57,E2 -27296.57} C_VEL
LIN {X 0,Y 98.936,Z 454.524,A -85,B 0,C 180,E1 -27297.376,E2 -27297.376} C_VEL
LIN {X 0,Y 100.995,Z 460.677,A -85,B 0,C 180,E1 -27298.467,E2 -27298.467} C_VEL
LIN {X 0,Y 96.184,Z 512.473,A -85,B 0,C 180,E1 -27304.016,E2 -27304.016} C_VEL
LIN {X 0,Y 94.908,Z 524.202,A -85,B 0,C 180,E1 -27305.835,E2 -27305.835} C_VEL
LIN {X 0,Y 92.976,Z 537.239,A -85,B 0,C 180,E1 -27308.644,E2 -27308.644} C_VEL
LIN {X 0,Y 90.708,Z 550.513,A -85,B 0,C 180,E1 -27312.606,E2 -27312.606} C_VEL
LIN {X 0,Y 88.721,Z 561.495,A -85,B 0,C 180,E1 -27316.903,E2 -27316.903} C_VEL
LIN {X 0,Y 86.81,Z 572.77,A -85,B 0,C 180,E1 -27322.615,E2 -27322.615} C_VEL
LIN {X 0,Y 85.669,Z 580.895,A -85,B 0,C 180,E1 -27327.775,E2 -27327.775} C_VEL
LIN {X 0,Y 84.967,Z 589.206,A -85,B 0,C 180,E1 -27334.262,E2 -27334.262} C_VEL
LIN {X 0,Y 84.601,Z 596.852,A -85,B 0,C 180,E1 -27341.848,E2 -27341.848} C_VEL
LIN {X 0,Y 85.596,Z 603.507,A -85,B 0,C 180,E1 -27350.12,E2 -27350.12} C_VEL
LIN {X 0,Y 87.981,Z 608.489,A -85,B 0,C 180,E1 -27357.711,E2 -27357.711} C_VEL
LIN {X 0,Y 91.635,Z 612.226,A -85,B 0,C 180,E1 -27364.485,E2 -27364.485} C_VEL
LIN {X 0,Y 98.374,Z 615.736,A -85,B 0,C 180,E1 -27372.376,E2 -27372.376} C_VEL
LIN {X 0,Y 102.501,Z 616.957,A -85,B 0,C 180,E1 -27375.918,E2 -27375.918} C_VEL
LIN {X 0,Y 112.054,Z 618.255,A -85,B 0,C 180,E1 -27382.106,E2 -27382.106} C_VEL
LIN {X 0,Y 122.966,Z 618.108,A -85,B 0,C 180,E1 -27387.208,E2 -27387.208} C_VEL
LIN {X 0,Y 129.196,Z 617.399,A -85,B 0,C 180,E1 -27389.508,E2 -27389.508} C_VEL
LIN {X 0,Y 141.415,Z 614.901,A -85,B 0,C 180,E1 -27393.139,E2 -27393.139} C_VEL
LIN {X 0,Y 130.67,Z 617.575,A -85,B 0,C 180,E1 -27396.227,E2 -27396.227} C_VEL
LIN {X 0,Y 119.549,Z 619.224,A -85,B 0,C 180,E1 -27400.168,E2 -27400.168} C_VEL
LIN {X 0,Y 109.765,Z 619.617,A -85,B 0,C 180,E1 -27405.234,E2 -27405.234} C_VEL
LIN {X 0,Y 101.016,Z 618.748,A -85,B 0,C 180,E1 -27411.24,E2 -27411.24} C_VEL
LIN {X 0,Y 93.853,Z 616.609,A -85,B 0,C 180,E1 -27418.394,E2 -27418.394} C_VEL
LIN {X 0,Y 88.935,Z 613.196,A -85,B 0,C 180,E1 -27426.733,E2 -27426.733} C_VEL
LIN {X 0,Y 86.428,Z 608.878,A -85,B 0,C 180,E1 -27435.135,E2 -27435.135} C_VEL
LIN {X 0,Y 84.42,Z 613.965,A -85,B 0,C 180,E1 -27442.833,E2 -27442.833} C_VEL
LIN {X 0,Y 84.125,Z 617.422,A -85,B 0,C 180,E1 -27450.006,E2 -27450.006} C_VEL
LIN {X 0,Y 83.987,Z 619.131,A -85,B 0,C 180,E1 -27454.806,E2 -27454.806} C_VEL
LIN {X 0,Y 85.053,Z 621.288,A -85,B 0,C 180,E1 -27464.359,E2 -27464.359} C_VEL
LIN {X 0,Y 88.163,Z 621.972,A -85,B 0,C 180,E1 -27473.496,E2 -27473.496} C_VEL
LIN {X 0,Y 93.547,Z 621.171,A -85,B 0,C 180,E1 -27481.735,E2 -27481.735} C_VEL
LIN {X 0,Y 100.707,Z 618.885,A -85,B 0,C 180,E1 -27488.915,E2 -27488.915} C_VEL
LIN {X 0,Y 109.218,Z 615.068,A -85,B 0,C 180,E1 -27495.065,E2 -27495.065} C_VEL
LIN {X 0,Y 116.373,Z 611.093,A -85,B 0,C 180,E1 -27499.023,E2 -27499.023} C_VEL
LIN {X 0,Y 121.11,Z 608.11,A -85,B 0,C 180,E1 -27501.142,E2 -27501.142} C_VEL
LIN {X 0,Y 124.704,Z 605.553,A -85,B 0,C 180,E1 -27502.974,E2 -27502.974} C_VEL
LIN {X 0,Y 129.565,Z 601.177,A -85,B 0,C 180,E1 -27506.335,E2 -27506.335} C_VEL
LIN {X 0,Y 134.548,Z 596.233,A -85,B 0,C 180,E1 -27509.361,E2 -27509.361} C_VEL
LIN {X 0,Y 138.186,Z 592.79,A -85,B 0,C 180,E1 -27510.662,E2 -27510.662} C_VEL
LIN {X 0,Y 146.436,Z 584.544,A -85,B 0,C 180,E1 -27512.615,E2 -27512.615} C_VEL
LIN {X 0,Y 155.013,Z 574.273,A -85,B 0,C 180,E1 -27514.309,E2 -27514.309} C_VEL
LIN {X 0,Y 162.168,Z 563.923,A -85,B 0,C 180,E1 -27515.525,E2 -27515.525} C_VEL
LIN {X 0,Y 168.625,Z 552.402,A -85,B 0,C 180,E1 -27516.487,E2 -27516.487} C_VEL
LIN {X 0,Y 173.891,Z 540.578,A -85,B 0,C 180,E1 -27517.175,E2 -27517.175} C_VEL
LIN {X 0,Y 178.189,Z 527.794,A -85,B 0,C 180,E1 -27517.731,E2 -27517.731} C_VEL
LIN {X 0,Y 178.415,Z 526.985,A -85,B 0,C 180,E1 -27517.753,E2 -27517.753} C_VEL
LIN {X 0,Y 178.443,Z 525.789,A -85,B 0,C 180,E1 -27519.239,E2 -27519.239} C_VEL
LIN {X 0,Y 178.435,Z 525.08,A -85,B 0,C 180,E1 -27521.634,E2 -27521.634} C_VEL
LIN {X 0,Y 178.711,Z 525.305,A -85,B 0,C 180,E1 -27524.41,E2 -27524.41} C_VEL
LIN {X 0,Y 178.673,Z 525.632,A -85,B 0,C 180,E1 -27524.649,E2 -27524.649} C_VEL
LIN {X 0,Y 174.897,Z 537.542,A -85,B 0,C 180,E1 -27525.232,E2 -27525.232} C_VEL
LIN {X 0,Y 169.517,Z 550.05,A -85,B 0,C 180,E1 -27526.069,E2 -27526.069} C_VEL
LIN {X 0,Y 163.405,Z 561.25,A -85,B 0,C 180,E1 -27527.124,E2 -27527.124} C_VEL
LIN {X 0,Y 156.28,Z 571.854,A -85,B 0,C 180,E1 -27528.476,E2 -27528.476} C_VEL
LIN {X 0,Y 147.985,Z 581.915,A -85,B 0,C 180,E1 -27530.226,E2 -27530.226} C_VEL
LIN {X 0,Y 140.135,Z 589.87,A -85,B 0,C 180,E1 -27532.117,E2 -27532.117} C_VEL
LIN {X 0,Y 130.554,Z 598.004,A -85,B 0,C 180,E1 -27534.845,E2 -27534.845} C_VEL
LIN {X 0,Y 122.121,Z 603.952,A -85,B 0,C 180,E1 -27537.735,E2 -27537.735} C_VEL
LIN {X 0,Y 112.509,Z 609.526,A -85,B 0,C 180,E1 -27541.755,E2 -27541.755} C_VEL
LIN {X 0,Y 105.858,Z 612.696,A -85,B 0,C 180,E1 -27545.167,E2 -27545.167} C_VEL
LIN {X 0,Y 99.649,Z 615.116,A -85,B 0,C 180,E1 -27549.081,E2 -27549.081} C_VEL
LIN {X 0,Y 93.977,Z 616.827,A -85,B 0,C 180,E1 -27553.522,E2 -27553.522} C_VEL
LIN {X 0,Y 88.934,Z 617.908,A -85,B 0,C 180,E1 -27558.488,E2 -27558.488} C_VEL
LIN {X 0,Y 84.166,Z 618.289,A -85,B 0,C 180,E1 -27564.678,E2 -27564.678} C_VEL
LIN {X 0,Y 80.393,Z 617.833,A -85,B 0,C 180,E1 -27571.637,E2 -27571.637} C_VEL
LIN {X 0,Y 77.772,Z 616.5,A -85,B 0,C 180,E1 -27579.241,E2 -27579.241} C_VEL
LIN {X 0,Y 76.202,Z 613.356,A -85,B 0,C 180,E1 -27589.781,E2 -27589.781} C_VEL
LIN {X 0,Y 76.79,Z 608.748,A -85,B 0,C 180,E1 -27599.769,E2 -27599.769} C_VEL
LIN {X 0,Y 78.246,Z 604.248,A -85,B 0,C 180,E1 -27606.946,E2 -27606.946} C_VEL
LIN {X 0,Y 80.936,Z 597.654,A -85,B 0,C 180,E1 -27614.894,E2 -27614.894} C_VEL
LIN {X 0,Y 84.409,Z 590.083,A -85,B 0,C 180,E1 -27621.711,E2 -27621.711} C_VEL
LIN {X 0,Y 88.708,Z 581.012,A -85,B 0,C 180,E1 -27627.724,E2 -27627.724} C_VEL
LIN {X 0,Y 93.385,Z 570.795,A -85,B 0,C 180,E1 -27632.69,E2 -27632.69} C_VEL
LIN {X 0,Y 97.863,Z 559.769,A -85,B 0,C 180,E1 -27636.642,E2 -27636.642} C_VEL
LIN {X 0,Y 102.248,Z 547.148,A -85,B 0,C 180,E1 -27639.889,E2 -27639.889} C_VEL
LIN {X 0,Y 105.601,Z 535.185,A -85,B 0,C 180,E1 -27642.111,E2 -27642.111} C_VEL
LIN {X 0,Y 108.35,Z 521.698,A -85,B 0,C 180,E1 -27643.852,E2 -27643.852} C_VEL
LIN {X 0,Y 110.324,Z 508.502,A -85,B 0,C 180,E1 -27644.854,E2 -27644.854} C_VEL
LIN {X 0,Y 113.367,Z 477.677,A -85,B 0,C 180,E1 -27646.595,E2 -27646.595} C_VEL
LIN {X 0,Y 112.695,Z 474.999,A -85,B 0,C 180,E1 -27647.161,E2 -27647.161} C_VEL
LIN {X 0,Y 110.293,Z 469.509,A -85,B 0,C 180,E1 -27648.853,E2 -27648.853} C_VEL
LIN {X 0,Y 105.522,Z 459.535,A -85,B 0,C 180,E1 -27652.513,E2 -27652.513} C_VEL
LIN {X 0,Y 102.532,Z 461.866,A -85,B 0,C 180,E1 -27654.044,E2 -27654.044} C_VEL
LIN {X 0,Y 101.542,Z 462.517,A -85,B 0,C 180,E1 -27654.589,E2 -27654.589} C_VEL
LIN {X 0,Y 97.74,Z 472.869,A -85,B 0,C 180,E1 -27655.724,E2 -27655.724} C_VEL
LIN {X 0,Y 95.318,Z 477.636,A -85,B 0,C 180,E1 -27656.763,E2 -27656.763} C_VEL
LIN {X 0,Y 94.069,Z 479.065,A -85,B 0,C 180,E1 -27657.476,E2 -27657.476} C_VEL
LIN {X 0,Y 93.323,Z 479.006,A -85,B 0,C 180,E1 -27658.051,E2 -27658.051} C_VEL
LIN {X 0,Y 92.825,Z 478.072,A -85,B 0,C 180,E1 -27658.576,E2 -27658.576} C_VEL
LIN {X 0,Y 92.675,Z 476.229,A -85,B 0,C 180,E1 -27658.971,E2 -27658.971} C_VEL
LIN {X 0,Y 88.864,Z 516.314,A -85,B 0,C 180,E1 -27663.795,E2 -27663.795} C_VEL
LIN {X 0,Y 87.148,Z 529.326,A -85,B 0,C 180,E1 -27666.249,E2 -27666.249} C_VEL
LIN {X 0,Y 85.001,Z 542.276,A -85,B 0,C 180,E1 -27669.648,E2 -27669.648} C_VEL
LIN {X 0,Y 82.988,Z 553.371,A -85,B 0,C 180,E1 -27673.561,E2 -27673.561} C_VEL
LIN {X 0,Y 80.977,Z 564.269,A -85,B 0,C 180,E1 -27678.564,E2 -27678.564} C_VEL
LIN {X 0,Y 79.32,Z 574.961,A -85,B 0,C 180,E1 -27684.835,E2 -27684.835} C_VEL
LIN {X 0,Y 78.303,Z 584.393,A -85,B 0,C 180,E1 -27691.887,E2 -27691.887} C_VEL
LIN {X 0,Y 77.784,Z 591.801,A -85,B 0,C 180,E1 -27698.812,E2 -27698.812} C_VEL
LIN {X 0,Y 78.132,Z 598.814,A -85,B 0,C 180,E1 -27707.004,E2 -27707.004} C_VEL
LIN {X 0,Y 79.828,Z 604.476,A -85,B 0,C 180,E1 -27714.949,E2 -27714.949} C_VEL
LIN {X 0,Y 82.908,Z 609.005,A -85,B 0,C 180,E1 -27722.429,E2 -27722.429} C_VEL
LIN {X 0,Y 87.359,Z 612.587,A -85,B 0,C 180,E1 -27729.259,E2 -27729.259} C_VEL
LIN {X 0,Y 95.316,Z 616.087,A -85,B 0,C 180,E1 -27737.153,E2 -27737.153} C_VEL
LIN {X 0,Y 105.08,Z 618.077,A -85,B 0,C 180,E1 -27743.659,E2 -27743.659} C_VEL
LIN {X 0,Y 116.218,Z 618.632,A -85,B 0,C 180,E1 -27748.932,E2 -27748.932} C_VEL
LIN {X 0,Y 127.291,Z 617.854,A -85,B 0,C 180,E1 -27752.767,E2 -27752.767} C_VEL
LIN {X 0,Y 126.611,Z 617.999,A -85,B 0,C 180,E1 -27753.639,E2 -27753.639} C_VEL
LIN {X 0,Y 115.11,Z 619.203,A -85,B 0,C 180,E1 -27757.474,E2 -27757.474} C_VEL
LIN {X 0,Y 104.849,Z 619.187,A -85,B 0,C 180,E1 -27762.504,E2 -27762.504} C_VEL
LIN {X 0,Y 95.624,Z 617.961,A -85,B 0,C 180,E1 -27768.596,E2 -27768.596} C_VEL
LIN {X 0,Y 87.971,Z 615.48,A -85,B 0,C 180,E1 -27776.005,E2 -27776.005} C_VEL
LIN {X 0,Y 82.597,Z 611.723,A -85,B 0,C 180,E1 -27784.829,E2 -27784.829} C_VEL
LIN {X 0,Y 79.873,Z 607.485,A -85,B 0,C 180,E1 -27793.39,E2 -27793.39} C_VEL
LIN {X 0,Y 77.424,Z 613.07,A -85,B 0,C 180,E1 -27802.181,E2 -27802.181} C_VEL
LIN {X 0,Y 77.076,Z 616.703,A -85,B 0,C 180,E1 -27810.007,E2 -27810.007} C_VEL
LIN {X 0,Y 76.932,Z 618.509,A -85,B 0,C 180,E1 -27815.248,E2 -27815.248} C_VEL
LIN {X 0,Y 77.291,Z 619.909,A -85,B 0,C 180,E1 -27820.485,E2 -27820.485} C_VEL
LIN {X 0,Y 79.64,Z 621.483,A -85,B 0,C 180,E1 -27830.677,E2 -27830.677} C_VEL
LIN {X 0,Y 84.366,Z 621.617,A -85,B 0,C 180,E1 -27839.995,E2 -27839.995} C_VEL
LIN {X 0,Y 91.21,Z 620.305,A -85,B 0,C 180,E1 -27848.062,E2 -27848.062} C_VEL
LIN {X 0,Y 99.677,Z 617.462,A -85,B 0,C 180,E1 -27854.843,E2 -27854.843} C_VEL
LIN {X 0,Y 109.302,Z 613.09,A -85,B 0,C 180,E1 -27860.503,E2 -27860.503} C_VEL
LIN {X 0,Y 117.28,Z 608.617,A -85,B 0,C 180,E1 -27864.004,E2 -27864.004} C_VEL
LIN {X 0,Y 126.999,Z 601.985,A -85,B 0,C 180,E1 -27867.564,E2 -27867.564} C_VEL
LIN {X 0,Y 137.352,Z 593.557,A -85,B 0,C 180,E1 -27870.448,E2 -27870.448} C_VEL
LIN {X 0,Y 138.186,Z 592.79,A -85,B 0,C 180,E1 -27870.662,E2 -27870.662} C_VEL
LIN {X 0,Y 141.861,Z 589.193,A -85,B 0,C 180,E1 -27871.864,E2 -27871.864} C_VEL
LIN {X 0,Y 147.092,Z 583.276,A -85,B 0,C 180,E1 -27874.254,E2 -27874.254} C_VEL
LIN {X 0,Y 152.139,Z 576.849,A -85,B 0,C 180,E1 -27876.374,E2 -27876.374} C_VEL
LIN {X 0,Y 155.405,Z 572.466,A -85,B 0,C 180,E1 -27877.178,E2 -27877.178} C_VEL
LIN {X 0,Y 162.717,Z 561.782,A -85,B 0,C 180,E1 -27878.228,E2 -27878.228} C_VEL
LIN {X 0,Y 168.943,Z 550.563,A -85,B 0,C 180,E1 -27879.024,E2 -27879.024} C_VEL
LIN {X 0,Y 173.992,Z 539.087,A -85,B 0,C 180,E1 -27879.592,E2 -27879.592} C_VEL
LIN {X 0,Y 176.39,Z 532.384,A -85,B 0,C 180,E1 -27879.841,E2 -27879.841} C_VEL
LIN {X 0,Y 176.479,Z 531.903,A -85,B 0,C 180,E1 -27882.546,E2 -27882.546} C_VEL
LIN {X 0,Y 171.943,Z 543.876,A -85,B 0,C 180,E1 -27883.235,E2 -27883.235} C_VEL
LIN {X 0,Y 166.311,Z 555.308,A -85,B 0,C 180,E1 -27884.063,E2 -27884.063} C_VEL
LIN {X 0,Y 160.048,Z 565.531,A -85,B 0,C 180,E1 -27885.041,E2 -27885.041} C_VEL
LIN {X 0,Y 152.818,Z 575.265,A -85,B 0,C 180,E1 -27886.306,E2 -27886.306} C_VEL
LIN {X 0,Y 144.676,Z 584.355,A -85,B 0,C 180,E1 -27887.87,E2 -27887.87} C_VEL
LIN {X 0,Y 135.637,Z 592.761,A -85,B 0,C 180,E1 -27889.913,E2 -27889.913} C_VEL
LIN {X 0,Y 127.764,Z 598.934,A -85,B 0,C 180,E1 -27891.973,E2 -27891.973} C_VEL
LIN {X 0,Y 120.066,Z 604.099,A -85,B 0,C 180,E1 -27894.358,E2 -27894.358} C_VEL
LIN {X 0,Y 112.608,Z 608.32,A -85,B 0,C 180,E1 -27897.027,E2 -27897.027} C_VEL
LIN {X 0,Y 101.966,Z 613.192,A -85,B 0,C 180,E1 -27901.835,E2 -27901.835} C_VEL
LIN {X 0,Y 92.228,Z 616.456,A -85,B 0,C 180,E1 -27907.809,E2 -27907.809} C_VEL
LIN {X 0,Y 84.368,Z 618.11,A -85,B 0,C 180,E1 -27914.472,E2 -27914.472} C_VEL
LIN {X 0,Y 78.941,Z 618.508,A -85,B 0,C 180,E1 -27920.862,E2 -27920.862} C_VEL
LIN {X 0,Y 73.421,Z 617.791,A -85,B 0,C 180,E1 -27930.502,E2 -27930.502} C_VEL
LIN {X 0,Y 70.969,Z 616.482,A -85,B 0,C 180,E1 -27937.594,E2 -27937.594} C_VEL
LIN {X 0,Y 69.173,Z 613.316,A -85,B 0,C 180,E1 -27948.727,E2 -27948.727} C_VEL
LIN {X 0,Y 69.669,Z 608.661,A -85,B 0,C 180,E1 -27959.701,E2 -27959.701} C_VEL
LIN {X 0,Y 71.381,Z 603.617,A -85,B 0,C 180,E1 -27968.325,E2 -27968.325} C_VEL
LIN {X 0,Y 74.109,Z 597.411,A -85,B 0,C 180,E1 -27976.278,E2 -27976.278} C_VEL
LIN {X 0,Y 77.803,Z 589.825,A -85,B 0,C 180,E1 -27983.538,E2 -27983.538} C_VEL
LIN {X 0,Y 82.499,Z 580.502,A -85,B 0,C 180,E1 -27989.994,E2 -27989.994} C_VEL
LIN {X 0,Y 87.487,Z 570.151,A -85,B 0,C 180,E1 -27995.179,E2 -27995.179} C_VEL
LIN {X 0,Y 92.348,Z 558.646,A -85,B 0,C 180,E1 -27999.31,E2 -27999.31} C_VEL
LIN {X 0,Y 96.925,Z 545.952,A -85,B 0,C 180,E1 -28002.558,E2 -28002.558} C_VEL
LIN {X 0,Y 100.294,Z 534.076,A -85,B 0,C 180,E1 -28004.71,E2 -28004.71} C_VEL
LIN {X 0,Y 103.127,Z 520.486,A -85,B 0,C 180,E1 -28006.424,E2 -28006.424} C_VEL
LIN {X 0,Y 105.037,Z 507.474,A -85,B 0,C 180,E1 -28007.369,E2 -28007.369} C_VEL
LIN {X 0,Y 107.954,Z 479.08,A -85,B 0,C 180,E1 -28008.991,E2 -28008.991} C_VEL
LIN {X 0,Y 106.378,Z 474.974,A -85,B 0,C 180,E1 -28010.259,E2 -28010.259} C_VEL
LIN {X 0,Y 104.177,Z 470.301,A -85,B 0,C 180,E1 -28012.023,E2 -28012.023} C_VEL
LIN {X 0,Y 103.895,Z 470.309,A -85,B 0,C 180,E1 -28012.186,E2 -28012.186} C_VEL
LIN {X 0,Y 100.587,Z 478.232,A -85,B 0,C 180,E1 -28013.219,E2 -28013.219} C_VEL
LIN {X 0,Y 98.018,Z 482.7,A -85,B 0,C 180,E1 -28014.258,E2 -28014.258} C_VEL
LIN {X 0,Y 95.931,Z 484.944,A -85,B 0,C 180,E1 -28015.337,E2 -28015.337} C_VEL
LIN {X 0,Y 94.848,Z 485.664,A -85,B 0,C 180,E1 -28015.987,E2 -28015.987} C_VEL
LIN {X 0,Y 89.875,Z 501.766,A -85,B 0,C 180,E1 -28017.355,E2 -28017.355} C_VEL
LIN {X 0,Y 86.257,Z 510.938,A -85,B 0,C 180,E1 -28018.841,E2 -28018.841} C_VEL
LIN {X 0,Y 84.381,Z 514.016,A -85,B 0,C 180,E1 -28019.906,E2 -28019.906} C_VEL
LIN {X 0,Y 83.328,Z 514.697,A -85,B 0,C 180,E1 -28020.703,E2 -28020.703} C_VEL
LIN {X 0,Y 82.518,Z 514.008,A -85,B 0,C 180,E1 -28021.602,E2 -28021.602} C_VEL
LIN {X 0,Y 82.306,Z 511.91,A -85,B 0,C 180,E1 -28022.232,E2 -28022.232} C_VEL
LIN {X 0,Y 80.664,Z 525.31,A -85,B 0,C 180,E1 -28024.687,E2 -28024.687} C_VEL
LIN {X 0,Y 78.582,Z 538.377,A -85,B 0,C 180,E1 -28028.088,E2 -28028.088} C_VEL
LIN {X 0,Y 76.302,Z 550.787,A -85,B 0,C 180,E1 -28032.534,E2 -28032.534} C_VEL
LIN {X 0,Y 74.276,Z 561.588,A -85,B 0,C 180,E1 -28037.61,E2 -28037.61} C_VEL
LIN {X 0,Y 72.471,Z 572.716,A -85,B 0,C 180,E1 -28044.417,E2 -28044.417} C_VEL
LIN {X 0,Y 71.471,Z 581.786,A -85,B 0,C 180,E1 -28051.444,E2 -28051.444} C_VEL
LIN {X 0,Y 71.057,Z 588.819,A -85,B 0,C 180,E1 -28058.228,E2 -28058.228} C_VEL
LIN {X 0,Y 71.283,Z 596.363,A -85,B 0,C 180,E1 -28067.183,E2 -28067.183} C_VEL
LIN {X 0,Y 72.64,Z 601.511,A -85,B 0,C 180,E1 -28074.447,E2 -28074.447} C_VEL
LIN {X 0,Y 75.628,Z 606.584,A -85,B 0,C 180,E1 -28082.663,E2 -28082.663} C_VEL
LIN {X 0,Y 81.906,Z 611.911,A -85,B 0,C 180,E1 -28092.387,E2 -28092.387} C_VEL
LIN {X 0,Y 89.577,Z 615.359,A -85,B 0,C 180,E1 -28099.716,E2 -28099.716} C_VEL
LIN {X 0,Y 98.184,Z 617.557,A -85,B 0,C 180,E1 -28105.434,E2 -28105.434} C_VEL
LIN {X 0,Y 109.599,Z 618.806,A -85,B 0,C 180,E1 -28110.863,E2 -28110.863} C_VEL
LIN {X 0,Y 114.026,Z 618.906,A -85,B 0,C 180,E1 -28112.508,E2 -28112.508} C_VEL
LIN {X 0,Y 113.809,Z 618.981,A -85,B 0,C 180,E1 -28113.614,E2 -28113.614} C_VEL
LIN {X 0,Y 105.424,Z 619.003,A -85,B 0,C 180,E1 -28116.882,E2 -28116.882} C_VEL
LIN {X 0,Y 95.191,Z 617.994,A -85,B 0,C 180,E1 -28122.421,E2 -28122.421} C_VEL
LIN {X 0,Y 86.154,Z 615.77,A -85,B 0,C 180,E1 -28129.271,E2 -28129.271} C_VEL
LIN {X 0,Y 79.013,Z 612.297,A -85,B 0,C 180,E1 -28137.753,E2 -28137.753} C_VEL
LIN {X 0,Y 74.411,Z 607.538,A -85,B 0,C 180,E1 -28147.811,E2 -28147.811} C_VEL
LIN {X 0,Y 73.504,Z 605.882,A -85,B 0,C 180,E1 -28151.182,E2 -28151.182} C_VEL
LIN {X 0,Y 70.945,Z 610.654,A -85,B 0,C 180,E1 -28158.58,E2 -28158.58} C_VEL
LIN {X 0,Y 70,Z 614.821,A -85,B 0,C 180,E1 -28167.13,E2 -28167.13} C_VEL
LIN {X 0,Y 70.007,Z 615.98,A -85,B 0,C 180,E1 -28170.007,E2 -28170.007} C_VEL
LIN {X 0,Y 69.897,Z 617.857,A -85,B 0,C 180,E1 -28175.778,E2 -28175.778} C_VEL
LIN {X 0,Y 71.356,Z 620.427,A -85,B 0,C 180,E1 -28187.194,E2 -28187.194} C_VEL
LIN {X 0,Y 75.304,Z 621.48,A -85,B 0,C 180,E1 -28197.824,E2 -28197.824} C_VEL
LIN {X 0,Y 81.798,Z 621.078,A -85,B 0,C 180,E1 -28206.98,E2 -28206.98} C_VEL
LIN {X 0,Y 90.111,Z 619.255,A -85,B 0,C 180,E1 -28214.59,E2 -28214.59} C_VEL
LIN {X 0,Y 99.722,Z 615.878,A -85,B 0,C 180,E1 -28220.834,E2 -28220.834} C_VEL
LIN {X 0,Y 107.65,Z 612.295,A -85,B 0,C 180,E1 -28224.701,E2 -28224.701} C_VEL
LIN {X 0,Y 116.12,Z 607.717,A -85,B 0,C 180,E1 -28227.93,E2 -28227.93} C_VEL
LIN {X 0,Y 124.888,Z 602.022,A -85,B 0,C 180,E1 -28230.729,E2 -28230.729} C_VEL
LIN {X 0,Y 135.59,Z 593.646,A -85,B 0,C 180,E1 -28233.403,E2 -28233.403} C_VEL
LIN {X 0,Y 144.955,Z 584.713,A -85,B 0,C 180,E1 -28235.386,E2 -28235.386} C_VEL
LIN {X 0,Y 153.76,Z 574.559,A -85,B 0,C 180,E1 -28236.913,E2 -28236.913} C_VEL
LIN {X 0,Y 155.405,Z 572.466,A -85,B 0,C 180,E1 -28237.178,E2 -28237.178} C_VEL
LIN {X 0,Y 157.525,Z 569.476,A -85,B 0,C 180,E1 -28237.765,E2 -28237.765} C_VEL
LIN {X 0,Y 163.304,Z 560.264,A -85,B 0,C 180,E1 -28240.635,E2 -28240.635} C_VEL
LIN {X 0,Y 165.189,Z 557.016,A -85,B 0,C 180,E1 -28241.084,E2 -28241.084} C_VEL
LIN {X 0,Y 166.299,Z 555.001,A -85,B 0,C 180,E1 -28241.556,E2 -28241.556} C_VEL
LIN {X 0,Y 159.21,Z 566.358,A -85,B 0,C 180,E1 -28242.524,E2 -28242.524} C_VEL
LIN {X 0,Y 151.062,Z 576.876,A -85,B 0,C 180,E1 -28243.791,E2 -28243.791} C_VEL
LIN {X 0,Y 142.881,Z 585.551,A -85,B 0,C 180,E1 -28245.184,E2 -28245.184} C_VEL
LIN {X 0,Y 133.886,Z 593.508,A -85,B 0,C 180,E1 -28246.974,E2 -28246.974} C_VEL
LIN {X 0,Y 123.297,Z 601.241,A -85,B 0,C 180,E1 -28249.513,E2 -28249.513} C_VEL
LIN {X 0,Y 112.24,Z 607.681,A -85,B 0,C 180,E1 -28252.806,E2 -28252.806} C_VEL
LIN {X 0,Y 103.406,Z 611.801,A -85,B 0,C 180,E1 -28256.103,E2 -28256.103} C_VEL
LIN {X 0,Y 94.968,Z 614.908,A -85,B 0,C 180,E1 -28260,E2 -28260} C_VEL
LIN {X 0,Y 84.856,Z 617.547,A -85,B 0,C 180,E1 -28266.294,E2 -28266.294} C_VEL
LIN {X 0,Y 78.856,Z 618.461,A -85,B 0,C 180,E1 -28271.341,E2 -28271.341} C_VEL
LIN {X 0,Y 73.574,Z 618.741,A -85,B 0,C 180,E1 -28277.188,E2 -28277.188} C_VEL
LIN {X 0,Y 69.005,Z 618.311,A -85,B 0,C 180,E1 -28284.042,E2 -28284.042} C_VEL
LIN {X 0,Y 65.16,Z 617.037,A -85,B 0,C 180,E1 -28292.636,E2 -28292.636} C_VEL
LIN {X 0,Y 62.737,Z 614.809,A -85,B 0,C 180,E1 -28302.233,E2 -28302.233} C_VEL
LIN {X 0,Y 62.012,Z 611.497,A -85,B 0,C 180,E1 -28312.499,E2 -28312.499} C_VEL
LIN {X 0,Y 63.102,Z 606.606,A -85,B 0,C 180,E1 -28323.536,E2 -28323.536} C_VEL
LIN {X 0,Y 65.387,Z 601.042,A -85,B 0,C 180,E1 -28332.767,E2 -28332.767} C_VEL
LIN {X 0,Y 68.812,Z 594.208,A -85,B 0,C 180,E1 -28341.18,E2 -28341.18} C_VEL
LIN {X 0,Y 73.251,Z 585.889,A -85,B 0,C 180,E1 -28348.618,E2 -28348.618} C_VEL
LIN {X 0,Y 78.753,Z 575.552,A -85,B 0,C 180,E1 -28355.113,E2 -28355.113} C_VEL
LIN {X 0,Y 83.675,Z 565.4,A -85,B 0,C 180,E1 -28359.664,E2 -28359.664} C_VEL
LIN {X 0,Y 88.515,Z 553.881,A -85,B 0,C 180,E1 -28363.338,E2 -28363.338} C_VEL
LIN {X 0,Y 92.883,Z 541.326,A -85,B 0,C 180,E1 -28366.195,E2 -28366.195} C_VEL
LIN {X 0,Y 96.342,Z 528.206,A -85,B 0,C 180,E1 -28368.255,E2 -28368.255} C_VEL
LIN {X 0,Y 98.83,Z 515.054,A -85,B 0,C 180,E1 -28369.6,E2 -28369.6} C_VEL
LIN {X 0,Y 102.128,Z 486.315,A -85,B 0,C 180,E1 -28371.305,E2 -28371.305} C_VEL
LIN {X 0,Y 101.994,Z 486.092,A -85,B 0,C 180,E1 -28371.41,E2 -28371.41} C_VEL
LIN {X 0,Y 99.049,Z 489.85,A -85,B 0,C 180,E1 -28372.718,E2 -28372.718} C_VEL
LIN {X 0,Y 98.307,Z 490.613,A -85,B 0,C 180,E1 -28373.072,E2 -28373.072} C_VEL
LIN {X 0,Y 93.508,Z 505.464,A -85,B 0,C 180,E1 -28374.212,E2 -28374.212} C_VEL
LIN {X 0,Y 89.77,Z 514.3,A -85,B 0,C 180,E1 -28375.474,E2 -28375.474} C_VEL
LIN {X 0,Y 87.176,Z 518.351,A -85,B 0,C 180,E1 -28376.572,E2 -28376.572} C_VEL
LIN {X 0,Y 85.061,Z 520.453,A -85,B 0,C 180,E1 -28377.787,E2 -28377.787} C_VEL
LIN {X 0,Y 83.374,Z 521.445,A -85,B 0,C 180,E1 -28378.962,E2 -28378.962} C_VEL
LIN {X 0,Y 79.885,Z 528.028,A -85,B 0,C 180,E1 -28380,E2 -28380} C_VEL
LIN {X 0,Y 77.805,Z 530.994,A -85,B 0,C 180,E1 -28380.893,E2 -28380.893} C_VEL
LIN {X 0,Y 76.357,Z 532.638,A -85,B 0,C 180,E1 -28381.637,E2 -28381.637} C_VEL
LIN {X 0,Y 75.013,Z 533.826,A -85,B 0,C 180,E1 -28382.517,E2 -28382.517} C_VEL
LIN {X 0,Y 72.448,Z 533.72,A -85,B 0,C 180,E1 -28385.585,E2 -28385.585} C_VEL
LIN {X 0,Y 72.374,Z 533.128,A -85,B 0,C 180,E1 -28385.996,E2 -28385.996} C_VEL
LIN {X 0,Y 69.809,Z 547.266,A -85,B 0,C 180,E1 -28390.968,E2 -28390.968} C_VEL
LIN {X 0,Y 67.523,Z 559.181,A -85,B 0,C 180,E1 -28396.756,E2 -28396.756} C_VEL
LIN {X 0,Y 65.657,Z 570.313,A -85,B 0,C 180,E1 -28403.933,E2 -28403.933} C_VEL
LIN {X 0,Y 64.661,Z 579.457,A -85,B 0,C 180,E1 -28411.446,E2 -28411.446} C_VEL
LIN {X 0,Y 64.274,Z 587.075,A -85,B 0,C 180,E1 -28419.183,E2 -28419.183} C_VEL
LIN {X 0,Y 64.599,Z 594.275,A -85,B 0,C 180,E1 -28428.238,E2 -28428.238} C_VEL
LIN {X 0,Y 66.316,Z 600.177,A -85,B 0,C 180,E1 -28436.962,E2 -28436.962} C_VEL
LIN {X 0,Y 70.948,Z 606.715,A -85,B 0,C 180,E1 -28447.924,E2 -28447.924} C_VEL
LIN {X 0,Y 76.779,Z 611.065,A -85,B 0,C 180,E1 -28455.938,E2 -28455.938} C_VEL
LIN {X 0,Y 86.106,Z 615.173,A -85,B 0,C 180,E1 -28464.085,E2 -28464.085} C_VEL
LIN {X 0,Y 97.14,Z 617.831,A -85,B 0,C 180,E1 -28470.427,E2 -28470.427} C_VEL
LIN {X 0,Y 101.911,Z 618.508,A -85,B 0,C 180,E1 -28472.526,E2 -28472.526} C_VEL
LIN {X 0,Y 101.329,Z 618.527,A -85,B 0,C 180,E1 -28473.674,E2 -28473.674} C_VEL
LIN {X 0,Y 90.587,Z 617.144,A -85,B 0,C 180,E1 -28479.13,E2 -28479.13} C_VEL
LIN {X 0,Y 80.979,Z 614.523,A -85,B 0,C 180,E1 -28486.038,E2 -28486.038} C_VEL
LIN {X 0,Y 73.265,Z 610.699,A -85,B 0,C 180,E1 -28494.871,E2 -28494.871} C_VEL
LIN {X 0,Y 67.7,Z 604.814,A -85,B 0,C 180,E1 -28507.098,E2 -28507.098} C_VEL
LIN {X 0,Y 67.261,Z 604.214,A -85,B 0,C 180,E1 -28508.557,E2 -28508.557} C_VEL
LIN {X 0,Y 64.062,Z 609.635,A -85,B 0,C 180,E1 -28517.334,E2 -28517.334} C_VEL
LIN {X 0,Y 62.95,Z 613.97,A -85,B 0,C 180,E1 -28526.808,E2 -28526.808} C_VEL
LIN {X 0,Y 62.811,Z 616.214,A -85,B 0,C 180,E1 -28533.215,E2 -28533.215} C_VEL
LIN {X 0,Y 63.384,Z 618.745,A -85,B 0,C 180,E1 -28542.821,E2 -28542.821} C_VEL
LIN {X 0,Y 66.521,Z 620.742,A -85,B 0,C 180,E1 -28555.008,E2 -28555.008} C_VEL
LIN {X 0,Y 72.401,Z 621.296,A -85,B 0,C 180,E1 -28565.63,E2 -28565.63} C_VEL
LIN {X 0,Y 80.495,Z 620.371,A -85,B 0,C 180,E1 -28574.314,E2 -28574.314} C_VEL
LIN {X 0,Y 90.169,Z 618.011,A -85,B 0,C 180,E1 -28581.216,E2 -28581.216} C_VEL
LIN {X 0,Y 98.116,Z 615.242,A -85,B 0,C 180,E1 -28585.469,E2 -28585.469} C_VEL
LIN {X 0,Y 106.62,Z 611.549,A -85,B 0,C 180,E1 -28588.98,E2 -28588.98} C_VEL
LIN {X 0,Y 115.494,Z 606.846,A -85,B 0,C 180,E1 -28591.935,E2 -28591.935} C_VEL
LIN {X 0,Y 124.736,Z 600.968,A -85,B 0,C 180,E1 -28594.363,E2 -28594.363} C_VEL
LIN {X 0,Y 134.199,Z 593.784,A -85,B 0,C 180,E1 -28596.425,E2 -28596.425} C_VEL
LIN {X 0,Y 143.827,Z 585.002,A -85,B 0,C 180,E1 -28598.198,E2 -28598.198} C_VEL
LIN {X 0,Y 152.829,Z 574.967,A -85,B 0,C 180,E1 -28599.557,E2 -28599.557} C_VEL
LIN {X 0,Y 161.12,Z 563.65,A -85,B 0,C 180,E1 -28600.618,E2 -28600.618} C_VEL
LIN {X 0,Y 165.189,Z 557.016,A -85,B 0,C 180,E1 -28601.084,E2 -28601.084} C_VEL
LIN {X 0,Y 164.114,Z 558.814,A -85,B 0,C 180,E1 -28601.348,E2 -28601.348} C_VEL
LIN {X 0,Y 160.919,Z 563.85,A -85,B 0,C 180,E1 -28601.522,E2 -28601.522} C_VEL
LIN {X 0,Y 153.697,Z 573.63,A -85,B 0,C 180,E1 -28601.49,E2 -28601.49} C_VEL
LIN {X 0,Y 148.843,Z 579.291,A -85,B 0,C 180,E1 -28601.339,E2 -28601.339} C_VEL
LIN {X 0,Y 141.136,Z 587.125,A -85,B 0,C 180,E1 -28600.731,E2 -28600.731} C_VEL
LIN {X 0,Y 138.473,Z 589.533,A -85,B 0,C 180,E1 -28600.37,E2 -28600.37} C_VEL
LIN {X 0,Y 128.322,Z 597.722,A -85,B 0,C 180,E1 -28598.612,E2 -28598.612} C_VEL
LIN {X 0,Y 118.659,Z 604.146,A -85,B 0,C 180,E1 -28596.651,E2 -28596.651} C_VEL
LIN {X 0,Y 109.294,Z 609.311,A -85,B 0,C 180,E1 -28594.2,E2 -28594.2} C_VEL
LIN {X 0,Y 100.146,Z 613.454,A -85,B 0,C 180,E1 -28591.319,E2 -28591.319} C_VEL
LIN {X 0,Y 91.421,Z 616.632,A -85,B 0,C 180,E1 -28587.749,E2 -28587.749} C_VEL
LIN {X 0,Y 80.605,Z 619.503,A -85,B 0,C 180,E1 -28581.704,E2 -28581.704} C_VEL
LIN {X 0,Y 70.931,Z 620.908,A -85,B 0,C 180,E1 -28573.924,E2 -28573.924} C_VEL
LIN {X 0,Y 63.061,Z 620.856,A -85,B 0,C 180,E1 -28563.875,E2 -28563.875} C_VEL
LIN {X 0,Y 57.947,Z 619.412,A -85,B 0,C 180,E1 -28551.346,E2 -28551.346} C_VEL
LIN {X 0,Y 56.49,Z 618.139,A -85,B 0,C 180,E1 -28544.417,E2 -28544.417} C_VEL
LIN {X 0,Y 55.773,Z 615.453,A -85,B 0,C 180,E1 -28533.622,E2 -28533.622} C_VEL
LIN {X 0,Y 55.917,Z 613.075,A -85,B 0,C 180,E1 -28526.406,E2 -28526.406} C_VEL
LIN {X 0,Y 57.22,Z 608.544,A -85,B 0,C 180,E1 -28515.789,E2 -28515.789} C_VEL
LIN {X 0,Y 61.386,Z 602.331,A -85,B 0,C 180,E1 -28505.263,E2 -28505.263} C_VEL
LIN {X 0,Y 66.07,Z 607.697,A -85,B 0,C 180,E1 -28494.204,E2 -28494.204} C_VEL
LIN {X 0,Y 71.65,Z 611.196,A -85,B 0,C 180,E1 -28486.647,E2 -28486.647} C_VEL
LIN {X 0,Y 81.036,Z 614.781,A -85,B 0,C 180,E1 -28478.7,E2 -28478.7} C_VEL
LIN {X 0,Y 86.327,Z 616.11,A -85,B 0,C 180,E1 -28475.511,E2 -28475.511} C_VEL
LIN {X 0,Y 90.704,Z 616.947,A -85,B 0,C 180,E1 -28472.845,E2 -28472.845} C_VEL
LIN {X 0,Y 79.366,Z 613.573,A -85,B 0,C 180,E1 -28466.28,E2 -28466.28} C_VEL
LIN {X 0,Y 69.78,Z 608.819,A -85,B 0,C 180,E1 -28457.586,E2 -28457.586} C_VEL
LIN {X 0,Y 64.073,Z 604.118,A -85,B 0,C 180,E1 -28449.234,E2 -28449.234} C_VEL
LIN {X 0,Y 59.704,Z 597.703,A -85,B 0,C 180,E1 -28438.313,E2 -28438.313} C_VEL
LIN {X 0,Y 57.753,Z 590.021,A -85,B 0,C 180,E1 -28426.746,E2 -28426.746} C_VEL
LIN {X 0,Y 57.664,Z 582.008,A -85,B 0,C 180,E1 -28416.664,E2 -28416.664} C_VEL
LIN {X 0,Y 58.238,Z 572.812,A -85,B 0,C 180,E1 -28407.627,E2 -28407.627} C_VEL
LIN {X 0,Y 59.683,Z 562.57,A -85,B 0,C 180,E1 -28399.634,E2 -28399.634} C_VEL
LIN {X 0,Y 61.706,Z 551.696,A -85,B 0,C 180,E1 -28393.095,E2 -28393.095} C_VEL
LIN {X 0,Y 62.693,Z 546.916,A -85,B 0,C 180,E1 -28390.703,E2 -28390.703} C_VEL
LIN {X 0,Y 63.168,Z 548.054,A -85,B 0,C 180,E1 -28388.847,E2 -28388.847} C_VEL
LIN {X 0,Y 65.303,Z 547.471,A -85,B 0,C 180,E1 -28386.179,E2 -28386.179} C_VEL
LIN {X 0,Y 67.957,Z 545.32,A -85,B 0,C 180,E1 -28384.171,E2 -28384.171} C_VEL
LIN {X 0,Y 71.205,Z 541.736,A -85,B 0,C 180,E1 -28382.593,E2 -28382.593} C_VEL
LIN {X 0,Y 76.234,Z 538.88,A -85,B 0,C 180,E1 -28378.859,E2 -28378.859} C_VEL
LIN {X 0,Y 79.199,Z 536.168,A -85,B 0,C 180,E1 -28377.452,E2 -28377.452} C_VEL
LIN {X 0,Y 82.544,Z 531.956,A -85,B 0,C 180,E1 -28376.27,E2 -28376.27} C_VEL
LIN {X 0,Y 85.934,Z 526.514,A -85,B 0,C 180,E1 -28375.383,E2 -28375.383} C_VEL
LIN {X 0,Y 89.266,Z 523.593,A -85,B 0,C 180,E1 -28373.757,E2 -28373.757} C_VEL
LIN {X 0,Y 92.568,Z 519.217,A -85,B 0,C 180,E1 -28372.582,E2 -28372.582} C_VEL
LIN {X 0,Y 93.062,Z 518.363,A -85,B 0,C 180,E1 -28372.43,E2 -28372.43} C_VEL
LIN {X 0,Y 93.253,Z 518.371,A -85,B 0,C 180,E1 -28372.308,E2 -28372.308} C_VEL
LIN {X 0,Y 90.674,Z 530.566,A -85,B 0,C 180,E1 -28370.938,E2 -28370.938} C_VEL
LIN {X 0,Y 86.981,Z 543.094,A -85,B 0,C 180,E1 -28368.85,E2 -28368.85} C_VEL
LIN {X 0,Y 82.577,Z 554.885,A -85,B 0,C 180,E1 -28366.051,E2 -28366.051} C_VEL
LIN {X 0,Y 77.896,Z 565.4,A -85,B 0,C 180,E1 -28362.567,E2 -28362.567} C_VEL
LIN {X 0,Y 72.461,Z 575.923,A -85,B 0,C 180,E1 -28357.672,E2 -28357.672} C_VEL
LIN {X 0,Y 67.134,Z 585.306,A -85,B 0,C 180,E1 -28351.492,E2 -28351.492} C_VEL
LIN {X 0,Y 62.268,Z 593.806,A -85,B 0,C 180,E1 -28343.511,E2 -28343.511} C_VEL
LIN {X 0,Y 58.448,Z 600.84,A -85,B 0,C 180,E1 -28334.148,E2 -28334.148} C_VEL
LIN {X 0,Y 56.209,Z 605.87,A -85,B 0,C 180,E1 -28325.151,E2 -28325.151} C_VEL
LIN {X 0,Y 54.991,Z 610.228,A -85,B 0,C 180,E1 -28314.881,E2 -28314.881} C_VEL
LIN {X 0,Y 55.802,Z 614.539,A -85,B 0,C 180,E1 -28300.902,E2 -28300.902} C_VEL
LIN {X 0,Y 59.262,Z 617.28,A -85,B 0,C 180,E1 -28288.319,E2 -28288.319} C_VEL
LIN {X 0,Y 65.905,Z 618.806,A -85,B 0,C 180,E1 -28276.285,E2 -28276.285} C_VEL
LIN {X 0,Y 71.355,Z 618.923,A -85,B 0,C 180,E1 -28269.919,E2 -28269.919} C_VEL
LIN {X 0,Y 77.556,Z 618.408,A -85,B 0,C 180,E1 -28264.503,E2 -28264.503} C_VEL
LIN {X 0,Y 84.344,Z 617.261,A -85,B 0,C 180,E1 -28259.96,E2 -28259.96} C_VEL
LIN {X 0,Y 95.605,Z 614.17,A -85,B 0,C 180,E1 -28254.334,E2 -28254.334} C_VEL
LIN {X 0,Y 106.986,Z 609.699,A -85,B 0,C 180,E1 -28250.209,E2 -28250.209} C_VEL
LIN {X 0,Y 117.759,Z 604.21,A -85,B 0,C 180,E1 -28247.182,E2 -28247.182} C_VEL
LIN {X 0,Y 127.342,Z 598.125,A -85,B 0,C 180,E1 -28244.991,E2 -28244.991} C_VEL
LIN {X 0,Y 137.781,Z 589.998,A -85,B 0,C 180,E1 -28243.032,E2 -28243.032} C_VEL
LIN {X 0,Y 145.47,Z 582.815,A -85,B 0,C 180,E1 -28241.812,E2 -28241.812} C_VEL
LIN {X 0,Y 144.719,Z 583.616,A -85,B 0,C 180,E1 -28241.268,E2 -28241.268} C_VEL
LIN {X 0,Y 138.473,Z 589.533,A -85,B 0,C 180,E1 -28240.37,E2 -28240.37} C_VEL
LIN {X 0,Y 134.964,Z 592.519,A -85,B 0,C 180,E1 -28240.205,E2 -28240.205} C_VEL
LIN {X 0,Y 130.304,Z 596.051,A -85,B 0,C 180,E1 -28240.763,E2 -28240.763} C_VEL
LIN {X 0,Y 121.77,Z 601.708,A -85,B 0,C 180,E1 -28242.639,E2 -28242.639} C_VEL
LIN {X 0,Y 110.006,Z 608.078,A -85,B 0,C 180,E1 -28245.194,E2 -28245.194} C_VEL
LIN {X 0,Y 100.249,Z 612.236,A -85,B 0,C 180,E1 -28247.859,E2 -28247.859} C_VEL
LIN {X 0,Y 90.817,Z 615.348,A -85,B 0,C 180,E1 -28251.097,E2 -28251.097} C_VEL
LIN {X 0,Y 81.885,Z 617.504,A -85,B 0,C 180,E1 -28255.077,E2 -28255.077} C_VEL
LIN {X 0,Y 73.553,Z 618.774,A -85,B 0,C 180,E1 -28260,E2 -28260} C_VEL
LIN {X 0,Y 63.903,Z 619.15,A -85,B 0,C 180,E1 -28268.129,E2 -28268.129} C_VEL
LIN {X 0,Y 58.254,Z 618.634,A -85,B 0,C 180,E1 -28275.139,E2 -28275.139} C_VEL
LIN {X 0,Y 53.615,Z 617.467,A -85,B 0,C 180,E1 -28283.402,E2 -28283.402} C_VEL
LIN {X 0,Y 49.872,Z 615.362,A -85,B 0,C 180,E1 -28294.312,E2 -28294.312} C_VEL
LIN {X 0,Y 47.985,Z 612.173,A -85,B 0,C 180,E1 -28307.082,E2 -28307.082} C_VEL
LIN {X 0,Y 48.385,Z 607.722,A -85,B 0,C 180,E1 -28320.636,E2 -28320.636} C_VEL
LIN {X 0,Y 50.986,Z 601.65,A -85,B 0,C 180,E1 -28333.987,E2 -28333.987} C_VEL
LIN {X 0,Y 55.255,Z 594.322,A -85,B 0,C 180,E1 -28345.212,E2 -28345.212} C_VEL
LIN {X 0,Y 60,Z 586.644,A -85,B 0,C 180,E1 -28353.349,E2 -28353.349} C_VEL
LIN {X 0,Y 65.796,Z 577.206,A -85,B 0,C 180,E1 -28360.176,E2 -28360.176} C_VEL
LIN {X 0,Y 71.888,Z 566.262,A -85,B 0,C 180,E1 -28365.588,E2 -28365.588} C_VEL
LIN {X 0,Y 77.084,Z 555.366,A -85,B 0,C 180,E1 -28369.292,E2 -28369.292} C_VEL
LIN {X 0,Y 81.864,Z 543.182,A -85,B 0,C 180,E1 -28372.199,E2 -28372.199} C_VEL
LIN {X 0,Y 82.826,Z 540.433,A -85,B 0,C 180,E1 -28372.713,E2 -28372.713} C_VEL
LIN {X 0,Y 81.668,Z 540.197,A -85,B 0,C 180,E1 -28373.671,E2 -28373.671} C_VEL
LIN {X 0,Y 79.176,Z 542.647,A -85,B 0,C 180,E1 -28374.513,E2 -28374.513} C_VEL
LIN {X 0,Y 77.662,Z 543.814,A -85,B 0,C 180,E1 -28375.182,E2 -28375.182} C_VEL
LIN {X 0,Y 72.009,Z 546.961,A -85,B 0,C 180,E1 -28378.55,E2 -28378.55} C_VEL
LIN {X 0,Y 68.143,Z 550.591,A -85,B 0,C 180,E1 -28380.159,E2 -28380.159} C_VEL
LIN {X 0,Y 65.934,Z 552.24,A -85,B 0,C 180,E1 -28381.488,E2 -28381.488} C_VEL
LIN {X 0,Y 63.161,Z 553.683,A -85,B 0,C 180,E1 -28383.794,E2 -28383.794} C_VEL
LIN {X 0,Y 61.037,Z 554.224,A -85,B 0,C 180,E1 -28386.292,E2 -28386.292} C_VEL
LIN {X 0,Y 55.849,Z 557.953,A -85,B 0,C 180,E1 -28390.97,E2 -28390.97} C_VEL
LIN {X 0,Y 53.915,Z 558.606,A -85,B 0,C 180,E1 -28394.196,E2 -28394.196} C_VEL
LIN {X 0,Y 53.37,Z 557.838,A -85,B 0,C 180,E1 -28396.912,E2 -28396.912} C_VEL
LIN {X 0,Y 53.31,Z 558.133,A -85,B 0,C 180,E1 -28397.495,E2 -28397.495} C_VEL
LIN {X 0,Y 51.662,Z 568.615,A -85,B 0,C 180,E1 -28405.965,E2 -28405.965} C_VEL
LIN {X 0,Y 50.963,Z 577.938,A -85,B 0,C 180,E1 -28415.561,E2 -28415.561} C_VEL
LIN {X 0,Y 50.982,Z 584.621,A -85,B 0,C 180,E1 -28423.995,E2 -28423.995} C_VEL
LIN {X 0,Y 52.329,Z 592.658,A -85,B 0,C 180,E1 -28436.149,E2 -28436.149} C_VEL
LIN {X 0,Y 55.667,Z 599.153,A -85,B 0,C 180,E1 -28447.252,E2 -28447.252} C_VEL
LIN {X 0,Y 60.861,Z 604.599,A -85,B 0,C 180,E1 -28456.779,E2 -28456.779} C_VEL
LIN {X 0,Y 69.944,Z 610.304,A -85,B 0,C 180,E1 -28466.633,E2 -28466.633} C_VEL
LIN {X 0,Y 78.498,Z 613.825,A -85,B 0,C 180,E1 -28472.492,E2 -28472.492} C_VEL
LIN {X 0,Y 76.872,Z 613.392,A -85,B 0,C 180,E1 -28474.645,E2 -28474.645} C_VEL
LIN {X 0,Y 66.813,Z 609.463,A -85,B 0,C 180,E1 -28482.593,E2 -28482.593} C_VEL
LIN {X 0,Y 58.983,Z 604.252,A -85,B 0,C 180,E1 -28493.444,E2 -28493.444} C_VEL
LIN {X 0,Y 55.505,Z 600.498,A -85,B 0,C 180,E1 -28501.663,E2 -28501.663} C_VEL
LIN {X 0,Y 51.547,Z 605.589,A -85,B 0,C 180,E1 -28510.082,E2 -28510.082} C_VEL
LIN {X 0,Y 49.164,Z 610.678,A -85,B 0,C 180,E1 -28521.792,E2 -28521.792} C_VEL
LIN {X 0,Y 48.867,Z 613.447,A -85,B 0,C 180,E1 -28530.011,E2 -28530.011} C_VEL
LIN {X 0,Y 48.889,Z 615.652,A -85,B 0,C 180,E1 -28538.276,E2 -28538.276} C_VEL
LIN {X 0,Y 51.41,Z 618.838,A -85,B 0,C 180,E1 -28554.223,E2 -28554.223} C_VEL
LIN {X 0,Y 57.289,Z 620.516,A -85,B 0,C 180,E1 -28567.846,E2 -28567.846} C_VEL
LIN {X 0,Y 65.985,Z 620.753,A -85,B 0,C 180,E1 -28578.219,E2 -28578.219} C_VEL
LIN {X 0,Y 76.406,Z 619.599,A -85,B 0,C 180,E1 -28585.889,E2 -28585.889} C_VEL
LIN {X 0,Y 87.841,Z 616.973,A -85,B 0,C 180,E1 -28591.664,E2 -28591.664} C_VEL
LIN {X 0,Y 100.082,Z 612.812,A -85,B 0,C 180,E1 -28595.92,E2 -28595.92} C_VEL
LIN {X 0,Y 109.581,Z 608.585,A -85,B 0,C 180,E1 -28598.441,E2 -28598.441} C_VEL
LIN {X 0,Y 120.962,Z 602.296,A -85,B 0,C 180,E1 -28600.732,E2 -28600.732} C_VEL
LIN {X 0,Y 125.938,Z 599.063,A -85,B 0,C 180,E1 -28601.578,E2 -28601.578} C_VEL
LIN {X 0,Y 125.705,Z 599.196,A -85,B 0,C 180,E1 -28601.899,E2 -28601.899} C_VEL
LIN {X 0,Y 121.77,Z 601.708,A -85,B 0,C 180,E1 -28602.639,E2 -28602.639} C_VEL
LIN {X 0,Y 116.824,Z 604.644,A -85,B 0,C 180,E1 -28603.304,E2 -28603.304} C_VEL
LIN {X 0,Y 107.97,Z 609.074,A -85,B 0,C 180,E1 -28603.682,E2 -28603.682} C_VEL
LIN {X 0,Y 98.829,Z 612.742,A -85,B 0,C 180,E1 -28604.206,E2 -28604.206} C_VEL
LIN {X 0,Y 93.475,Z 614.472,A -85,B 0,C 180,E1 -28605.242,E2 -28605.242} C_VEL
LIN {X 0,Y 86.395,Z 616.443,A -85,B 0,C 180,E1 -28607.491,E2 -28607.491} C_VEL
LIN {X 0,Y 78.35,Z 618.048,A -85,B 0,C 180,E1 -28610.682,E2 -28610.682} C_VEL
LIN {X 0,Y 70.591,Z 619.06,A -85,B 0,C 180,E1 -28614.689,E2 -28614.689} C_VEL
LIN {X 0,Y 62.795,Z 619.407,A -85,B 0,C 180,E1 -28620.001,E2 -28620.001} C_VEL
LIN {X 0,Y 55.239,Z 618.987,A -85,B 0,C 180,E1 -28627.31,E2 -28627.31} C_VEL
LIN {X 0,Y 48.8,Z 617.739,A -85,B 0,C 180,E1 -28636.741,E2 -28636.741} C_VEL
LIN {X 0,Y 43.948,Z 615.615,A -85,B 0,C 180,E1 -28648.67,E2 -28648.67} C_VEL
LIN {X 0,Y 40.919,Z 611.575,A -85,B 0,C 180,E1 -28666.588,E2 -28666.588} C_VEL
LIN {X 0,Y 41.416,Z 606.982,A -85,B 0,C 180,E1 -28682.168,E2 -28682.168} C_VEL
LIN {X 0,Y 43.735,Z 602.015,A -85,B 0,C 180,E1 -28694.623,E2 -28694.623} C_VEL
LIN {X 0,Y 48.475,Z 594.477,A -85,B 0,C 180,E1 -28707.791,E2 -28707.791} C_VEL
LIN {X 0,Y 54.224,Z 585.953,A -85,B 0,C 180,E1 -28717.437,E2 -28717.437} C_VEL
LIN {X 0,Y 60.386,Z 576.646,A -85,B 0,C 180,E1 -28724.31,E2 -28724.31} C_VEL
LIN {X 0,Y 66.699,Z 565.992,A -85,B 0,C 180,E1 -28729.573,E2 -28729.573} C_VEL
LIN {X 0,Y 72.366,Z 554.682,A -85,B 0,C 180,E1 -28733.317,E2 -28733.317} C_VEL
LIN {X 0,Y 72.838,Z 553.604,A -85,B 0,C 180,E1 -28733.62,E2 -28733.62} C_VEL
LIN {X 0,Y 72.574,Z 552.361,A -85,B 0,C 180,E1 -28734.652,E2 -28734.652} C_VEL
LIN {X 0,Y 68.459,Z 555.744,A -85,B 0,C 180,E1 -28736.066,E2 -28736.066} C_VEL
LIN {X 0,Y 64.008,Z 558.385,A -85,B 0,C 180,E1 -28738.549,E2 -28738.549} C_VEL
LIN {X 0,Y 58.7,Z 560.626,A -85,B 0,C 180,E1 -28743.059,E2 -28743.059} C_VEL
LIN {X 0,Y 55.857,Z 562.488,A -85,B 0,C 180,E1 -28745.13,E2 -28745.13} C_VEL
LIN {X 0,Y 53.293,Z 563.798,A -85,B 0,C 180,E1 -28747.697,E2 -28747.697} C_VEL
LIN {X 0,Y 49.148,Z 565.223,A -85,B 0,C 180,E1 -28754.357,E2 -28754.357} C_VEL
LIN {X 0,Y 46.909,Z 566.727,A -85,B 0,C 180,E1 -28757.613,E2 -28757.613} C_VEL
LIN {X 0,Y 45.218,Z 567.459,A -85,B 0,C 180,E1 -28761.558,E2 -28761.558} C_VEL
LIN {X 0,Y 44.711,Z 567.041,A -85,B 0,C 180,E1 -28765.262,E2 -28765.262} C_VEL
LIN {X 0,Y 44.822,Z 566.678,A -85,B 0,C 180,E1 -28766.546,E2 -28766.546} C_VEL
LIN {X 0,Y 44.264,Z 575.542,A -85,B 0,C 180,E1 -28776.612,E2 -28776.612} C_VEL
LIN {X 0,Y 44.448,Z 581.733,A -85,B 0,C 180,E1 -28785.123,E2 -28785.123} C_VEL
LIN {X 0,Y 46.335,Z 590.774,A -85,B 0,C 180,E1 -28799.999,E2 -28799.999} C_VEL
LIN {X 0,Y 51.36,Z 598.696,A -85,B 0,C 180,E1 -28814.158,E2 -28814.158} C_VEL
LIN {X 0,Y 58.635,Z 604.822,A -85,B 0,C 180,E1 -28824.803,E2 -28824.803} C_VEL
LIN {X 0,Y 66.511,Z 609.307,A -85,B 0,C 180,E1 -28831.892,E2 -28831.892} C_VEL
LIN {X 0,Y 67.596,Z 609.846,A -85,B 0,C 180,E1 -28833.734,E2 -28833.734} C_VEL
LIN {X 0,Y 57.723,Z 604.905,A -85,B 0,C 180,E1 -28843.084,E2 -28843.084} C_VEL
LIN {X 0,Y 50.267,Z 598.311,A -85,B 0,C 180,E1 -28856.91,E2 -28856.91} C_VEL
LIN {X 0,Y 45.775,Z 603.31,A -85,B 0,C 180,E1 -28865.038,E2 -28865.038} C_VEL
LIN {X 0,Y 42.83,Z 607.937,A -85,B 0,C 180,E1 -28875.764,E2 -28875.764} C_VEL
LIN {X 0,Y 41.827,Z 612.482,A -85,B 0,C 180,E1 -28890.012,E2 -28890.012} C_VEL
LIN {X 0,Y 41.929,Z 614.846,A -85,B 0,C 180,E1 -28899.662,E2 -28899.662} C_VEL
LIN {X 0,Y 45.043,Z 618.219,A -85,B 0,C 180,E1 -28917.923,E2 -28917.923} C_VEL
LIN {X 0,Y 51.855,Z 620.108,A -85,B 0,C 180,E1 -28932.674,E2 -28932.674} C_VEL
LIN {X 0,Y 61.47,Z 620.6,A -85,B 0,C 180,E1 -28943.175,E2 -28943.175} C_VEL
LIN {X 0,Y 72.652,Z 619.644,A -85,B 0,C 180,E1 -28950.544,E2 -28950.544} C_VEL
LIN {X 0,Y 84.702,Z 617.296,A -85,B 0,C 180,E1 -28955.896,E2 -28955.896} C_VEL
LIN {X 0,Y 94.187,Z 614.526,A -85,B 0,C 180,E1 -28958.877,E2 -28958.877} C_VEL
LIN {X 0,Y 103.938,Z 610.836,A -85,B 0,C 180,E1 -28961.212,E2 -28961.212} C_VEL
LIN {X 0,Y 105.121,Z 610.295,A -85,B 0,C 180,E1 -28962.266,E2 -28962.266} C_VEL
LIN {X 0,Y 93.475,Z 614.472,A -85,B 0,C 180,E1 -28965.242,E2 -28965.242} C_VEL
LIN {X 0,Y 88.072,Z 616.026,A -85,B 0,C 180,E1 -28966.447,E2 -28966.447} C_VEL
LIN {X 0,Y 78.527,Z 618.038,A -85,B 0,C 180,E1 -28967.669,E2 -28967.669} C_VEL
LIN {X 0,Y 68.958,Z 619.316,A -85,B 0,C 180,E1 -28969.303,E2 -28969.303} C_VEL
LIN {X 0,Y 63.618,Z 619.594,A -85,B 0,C 180,E1 -28971.428,E2 -28971.428} C_VEL
LIN {X 0,Y 52.061,Z 619.205,A -85,B 0,C 180,E1 -28980.001,E2 -28980.001} C_VEL
LIN {X 0,Y 43.051,Z 617.554,A -85,B 0,C 180,E1 -28991.568,E2 -28991.568} C_VEL
LIN {X 0,Y 36.242,Z 614.372,A -85,B 0,C 180,E1 -29009.204,E2 -29009.204} C_VEL
LIN {X 0,Y 33.711,Z 609.659,A -85,B 0,C 180,E1 -29031.266,E2 -29031.266} C_VEL
LIN {X 0,Y 34.72,Z 605.644,A -85,B 0,C 180,E1 -29046.103,E2 -29046.103} C_VEL
LIN {X 0,Y 38.25,Z 599.593,A -85,B 0,C 180,E1 -29062.066,E2 -29062.066} C_VEL
LIN {X 0,Y 43.573,Z 592.256,A -85,B 0,C 180,E1 -29074.614,E2 -29074.614} C_VEL
LIN {X 0,Y 49.994,Z 583.651,A -85,B 0,C 180,E1 -29083.885,E2 -29083.885} C_VEL
LIN {X 0,Y 57.092,Z 573.354,A -85,B 0,C 180,E1 -29090.717,E2 -29090.717} C_VEL
LIN {X 0,Y 62.2,Z 565.025,A -85,B 0,C 180,E1 -29094.409,E2 -29094.409} C_VEL
LIN {X 0,Y 62.136,Z 564.258,A -85,B 0,C 180,E1 -29095.194,E2 -29095.194} C_VEL
LIN {X 0,Y 56.382,Z 566.778,A -85,B 0,C 180,E1 -29099.241,E2 -29099.241} C_VEL
LIN {X 0,Y 51.334,Z 569.209,A -85,B 0,C 180,E1 -29103.192,E2 -29103.192} C_VEL
LIN {X 0,Y 46.088,Z 570.989,A -85,B 0,C 180,E1 -29110.318,E2 -29110.318} C_VEL
LIN {X 0,Y 41.768,Z 572.97,A -85,B 0,C 180,E1 -29117.696,E2 -29117.696} C_VEL
LIN {X 0,Y 38.782,Z 574.145,A -85,B 0,C 180,E1 -29127.066,E2 -29127.066} C_VEL
LIN {X 0,Y 37.236,Z 575.011,A -85,B 0,C 180,E1 -29137.821,E2 -29137.821} C_VEL
LIN {X 0,Y 37.693,Z 574.428,A -85,B 0,C 180,E1 -29140.282,E2 -29140.282} C_VEL
LIN {X 0,Y 38.175,Z 580.175,A -85,B 0,C 180,E1 -29149.39,E2 -29149.39} C_VEL
LIN {X 0,Y 40.665,Z 588.757,A -85,B 0,C 180,E1 -29164.956,E2 -29164.956} C_VEL
LIN {X 0,Y 46.561,Z 596.773,A -85,B 0,C 180,E1 -29179.853,E2 -29179.853} C_VEL
LIN {X 0,Y 54.902,Z 603.372,A -85,B 0,C 180,E1 -29190.799,E2 -29190.799} C_VEL
LIN {X 0,Y 56.538,Z 604.371,A -85,B 0,C 180,E1 -29192.305,E2 -29192.305} C_VEL
LIN {X 0,Y 55.126,Z 603.659,A -85,B 0,C 180,E1 -29195.892,E2 -29195.892} C_VEL
LIN {X 0,Y 45.884,Z 596.709,A -85,B 0,C 180,E1 -29209.982,E2 -29209.982} C_VEL
LIN {X 0,Y 45.284,Z 596.155,A -85,B 0,C 180,E1 -29211.322,E2 -29211.322} C_VEL
LIN {X 0,Y 40.503,Z 600.822,A -85,B 0,C 180,E1 -29218.646,E2 -29218.646} C_VEL
LIN {X 0,Y 36.084,Z 606.723,A -85,B 0,C 180,E1 -29233.028,E2 -29233.028} C_VEL
LIN {X 0,Y 34.793,Z 611.479,A -85,B 0,C 180,E1 -29250.015,E2 -29250.015} C_VEL
LIN {X 0,Y 35.493,Z 614.994,A -85,B 0,C 180,E1 -29267.294,E2 -29267.294} C_VEL
LIN {X 0,Y 38.927,Z 617.575,A -85,B 0,C 180,E1 -29282.81,E2 -29282.81} C_VEL
LIN {X 0,Y 46.877,Z 619.661,A -85,B 0,C 180,E1 -29298.574,E2 -29298.574} C_VEL
LIN {X 0,Y 57.487,Z 620.375,A -85,B 0,C 180,E1 -29308.863,E2 -29308.863} C_VEL
LIN {X 0,Y 69.429,Z 619.7,A -85,B 0,C 180,E1 -29315.665,E2 -29315.665} C_VEL
LIN {X 0,Y 82.067,Z 617.566,A -85,B 0,C 180,E1 -29320.41,E2 -29320.41} C_VEL
LIN {X 0,Y 83.554,Z 617.23,A -85,B 0,C 180,E1 -29320.861,E2 -29320.861} C_VEL
LIN {X 0,Y 86.149,Z 616.581,A -85,B 0,C 180,E1 -29322.389,E2 -29322.389} C_VEL
LIN {X 0,Y 79.117,Z 617.999,A -85,B 0,C 180,E1 -29324.545,E2 -29324.545} C_VEL
LIN {X 0,Y 69.601,Z 619.249,A -85,B 0,C 180,E1 -29328.349,E2 -29328.349} C_VEL
LIN {X 0,Y 63.618,Z 619.594,A -85,B 0,C 180,E1 -29331.428,E2 -29331.428} C_VEL
LIN {X 0,Y 58.365,Z 619.639,A -85,B 0,C 180,E1 -29333.955,E2 -29333.955} C_VEL
LIN {X 0,Y 49.072,Z 619.142,A -85,B 0,C 180,E1 -29337.561,E2 -29337.561} C_VEL
LIN {X 0,Y 41.801,Z 618.139,A -85,B 0,C 180,E1 -29341.418,E2 -29341.418} C_VEL
LIN {X 0,Y 37.006,Z 617.069,A -85,B 0,C 180,E1 -29346.251,E2 -29346.251} C_VEL
LIN {X 0,Y 35.656,Z 616.66,A -85,B 0,C 180,E1 -29348.453,E2 -29348.453} C_VEL
LIN {X 0,Y 28.613,Z 612.974,A -85,B 0,C 180,E1 -29369.424,E2 -29369.424} C_VEL
LIN {X 0,Y 26.649,Z 608.732,A -85,B 0,C 180,E1 -29392.297,E2 -29392.297} C_VEL
LIN {X 0,Y 28.269,Z 604.152,A -85,B 0,C 180,E1 -29411.883,E2 -29411.883} C_VEL
LIN {X 0,Y 32.887,Z 597.738,A -85,B 0,C 180,E1 -29429.984,E2 -29429.984} C_VEL
LIN {X 0,Y 39.377,Z 589.937,A -85,B 0,C 180,E1 -29442.877,E2 -29442.877} C_VEL
LIN {X 0,Y 47.034,Z 580.425,A -85,B 0,C 180,E1 -29451.923,E2 -29451.923} C_VEL
LIN {X 0,Y 51.445,Z 574.468,A -85,B 0,C 180,E1 -29455.558,E2 -29455.558} C_VEL
LIN {X 0,Y 49.77,Z 574.322,A -85,B 0,C 180,E1 -29457.933,E2 -29457.933} C_VEL
LIN {X 0,Y 43.179,Z 576.31,A -85,B 0,C 180,E1 -29465.527,E2 -29465.527} C_VEL
LIN {X 0,Y 38.366,Z 578.199,A -85,B 0,C 180,E1 -29472.883,E2 -29472.883} C_VEL
LIN {X 0,Y 34.254,Z 579.545,A -85,B 0,C 180,E1 -29485.127,E2 -29485.127} C_VEL
LIN {X 0,Y 32.782,Z 580.188,A -85,B 0,C 180,E1 -29494.609,E2 -29494.609} C_VEL
LIN {X 0,Y 31.404,Z 581.767,A -85,B 0,C 180,E1 -29507.067,E2 -29507.067} C_VEL
LIN {X 0,Y 32.369,Z 582.539,A -85,B 0,C 180,E1 -29519.999,E2 -29519.999} C_VEL
LIN {X 0,Y 33.375,Z 582.361,A -85,B 0,C 180,E1 -29523.017,E2 -29523.017} C_VEL
LIN {X 0,Y 37.888,Z 590.037,A -85,B 0,C 180,E1 -29538.349,E2 -29538.349} C_VEL
LIN {X 0,Y 46.092,Z 597.82,A -85,B 0,C 180,E1 -29551.777,E2 -29551.777} C_VEL
LIN {X 0,Y 47.547,Z 598.865,A -85,B 0,C 180,E1 -29553.407,E2 -29553.407} C_VEL
LIN {X 0,Y 44.591,Z 596.791,A -85,B 0,C 180,E1 -29558.016,E2 -29558.016} C_VEL
LIN {X 0,Y 40.995,Z 593.793,A -85,B 0,C 180,E1 -29564.402,E2 -29564.402} C_VEL
LIN {X 0,Y 34.75,Z 599.339,A -85,B 0,C 180,E1 -29572.666,E2 -29572.666} C_VEL
LIN {X 0,Y 29.45,Z 605.458,A -85,B 0,C 180,E1 -29589.044,E2 -29589.044} C_VEL
LIN {X 0,Y 27.762,Z 610.414,A -85,B 0,C 180,E1 -29610.019,E2 -29610.019} C_VEL
LIN {X 0,Y 28.836,Z 614.11,A -85,B 0,C 180,E1 -29631.463,E2 -29631.463} C_VEL
LIN {X 0,Y 33.199,Z 616.846,A -85,B 0,C 180,E1 -29649.445,E2 -29649.445} C_VEL
LIN {X 0,Y 42.511,Z 619.199,A -85,B 0,C 180,E1 -29665.773,E2 -29665.773} C_VEL
LIN {X 0,Y 54.152,Z 620.121,A -85,B 0,C 180,E1 -29675.318,E2 -29675.318} C_VEL
LIN {X 0,Y 66.813,Z 619.667,A -85,B 0,C 180,E1 -29681.232,E2 -29681.232} C_VEL
LIN {X 0,Y 68.777,Z 619.492,A -85,B 0,C 180,E1 -29682.149,E2 -29682.149} C_VEL
LIN {X 0,Y 57.734,Z 619.865,A -85,B 0,C 180,E1 -29686.903,E2 -29686.903} C_VEL
LIN {X 0,Y 49.691,Z 619.403,A -85,B 0,C 180,E1 -29691.973,E2 -29691.973} C_VEL
LIN {X 0,Y 41.299,Z 618.154,A -85,B 0,C 180,E1 -29700.001,E2 -29700.001} C_VEL
LIN {X 0,Y 35.656,Z 616.66,A -85,B 0,C 180,E1 -29708.453,E2 -29708.453} C_VEL
LIN {X 0,Y 31.671,Z 615.346,A -85,B 0,C 180,E1 -29715.534,E2 -29715.534} C_VEL
LIN {X 0,Y 24.958,Z 612.354,A -85,B 0,C 180,E1 -29729.116,E2 -29729.116} C_VEL
LIN {X 0,Y 20.335,Z 608.53,A -85,B 0,C 180,E1 -29749.534,E2 -29749.534} C_VEL
LIN {X 0,Y 20.135,Z 605.907,A -85,B 0,C 180,E1 -29764.719,E2 -29764.719} C_VEL
LIN {X 0,Y 24.43,Z 599.924,A -85,B 0,C 180,E1 -29789.979,E2 -29789.979} C_VEL
LIN {X 0,Y 31.36,Z 592.559,A -85,B 0,C 180,E1 -29806.251,E2 -29806.251} C_VEL
LIN {X 0,Y 39.081,Z 584.133,A -85,B 0,C 180,E1 -29815.949,E2 -29815.949} C_VEL
LIN {X 0,Y 40.548,Z 582.414,A -85,B 0,C 180,E1 -29817.273,E2 -29817.273} C_VEL
LIN {X 0,Y 40.472,Z 581.348,A -85,B 0,C 180,E1 -29819.742,E2 -29819.742} C_VEL
LIN {X 0,Y 35.006,Z 583.203,A -85,B 0,C 180,E1 -29827.015,E2 -29827.015} C_VEL
LIN {X 0,Y 28.191,Z 585.087,A -85,B 0,C 180,E1 -29850.091,E2 -29850.091} C_VEL
LIN {X 0,Y 26.364,Z 586.574,A -85,B 0,C 180,E1 -29864.538,E2 -29864.538} C_VEL
LIN {X 0,Y 27.118,Z 587.346,A -85,B 0,C 180,E1 -29879.999,E2 -29879.999} C_VEL
LIN {X 0,Y 29.174,Z 588.991,A -85,B 0,C 180,E1 -29895.573,E2 -29895.573} C_VEL
LIN {X 0,Y 32.419,Z 589.851,A -85,B 0,C 180,E1 -29905.694,E2 -29905.694} C_VEL
LIN {X 0,Y 35.861,Z 589.786,A -85,B 0,C 180,E1 -29910.551,E2 -29910.551} C_VEL
LIN {X 0,Y 37.988,Z 591.716,A -85,B 0,C 180,E1 -29913.711,E2 -29913.711} C_VEL
LIN {X 0,Y 37.359,Z 591.311,A -85,B 0,C 180,E1 -29916.114,E2 -29916.114} C_VEL
LIN {X 0,Y 31.141,Z 596.361,A -85,B 0,C 180,E1 -29922.102,E2 -29922.102} C_VEL
LIN {X 0,Y 24.878,Z 602.09,A -85,B 0,C 180,E1 -29935.623,E2 -29935.623} C_VEL
LIN {X 0,Y 20.976,Z 607.675,A -85,B 0,C 180,E1 -29960.381,E2 -29960.381} C_VEL
LIN {X 0,Y 20.826,Z 610.69,A -85,B 0,C 180,E1 -29979.74,E2 -29979.74} C_VEL
LIN {X 0,Y 23.931,Z 614.25,A -85,B 0,C 180,E1 -30005.996,E2 -30005.996} C_VEL
LIN {X 0,Y 33.195,Z 617.53,A -85,B 0,C 180,E1 -30027.902,E2 -30027.902} C_VEL
LIN {X 0,Y 45.176,Z 619.415,A -85,B 0,C 180,E1 -30039.006,E2 -30039.006} C_VEL
LIN {X 0,Y 48.654,Z 619.622,A -85,B 0,C 180,E1 -30043.209,E2 -30043.209} C_VEL
LIN {X 0,Y 35.379,Z 617.556,A -85,B 0,C 180,E1 -30053.455,E2 -30053.455} C_VEL
LIN {X 0,Y 25.455,Z 614.265,A -85,B 0,C 180,E1 -30070.702,E2 -30070.702} C_VEL
LIN {X 0,Y 19.727,Z 609.164,A -85,B 0,C 180,E1 -30104.521,E2 -30104.521} C_VEL
LIN {X 0,Y 20.135,Z 605.907,A -85,B 0,C 180,E1 -30124.719,E2 -30124.719} C_VEL
LIN {X 0,Y 20.458,Z 604.064,A -85,B 0,C 180,E1 -30134.534,E2 -30134.534} C_VEL
LIN {X 0,Y 20.417,Z 600.734,A -85,B 0,C 180,E1 -30151.032,E2 -30151.032} C_VEL
LIN {X 0,Y 21.732,Z 597.131,A -85,B 0,C 180,E1 -30166.344,E2 -30166.344} C_VEL
LIN {X 0,Y 23.813,Z 594.742,A -85,B 0,C 180,E1 -30172.573,E2 -30172.573} C_VEL
LIN {X 0,Y 30.153,Z 588.809,A -85,B 0,C 180,E1 -30180.759,E2 -30180.759} C_VEL
LIN {X 0,Y 28.542,Z 588.61,A -85,B 0,C 180,E1 -30186.047,E2 -30186.047} C_VEL
LIN {X 0,Y 23.634,Z 589.689,A -85,B 0,C 180,E1 -30203.504,E2 -30203.504} C_VEL
LIN {X 0,Y 21.168,Z 591.101,A -85,B 0,C 180,E1 -30220.607,E2 -30220.607} C_VEL
LIN {X 0,Y 21.609,Z 591.877,A -85,B 0,C 180,E1 -30239.998,E2 -30239.998} C_VEL
LIN {X 0,Y 26.817,Z 594.079,A -85,B 0,C 180,E1 -30269.036,E2 -30269.036} C_VEL
LIN {X 0,Y 26.18,Z 595.255,A -85,B 0,C 180,E1 -30272.135,E2 -30272.135} C_VEL
